Yaskawa INFORM job: A_ROOF_SIDE_0617_2_PAINT_23.JBI

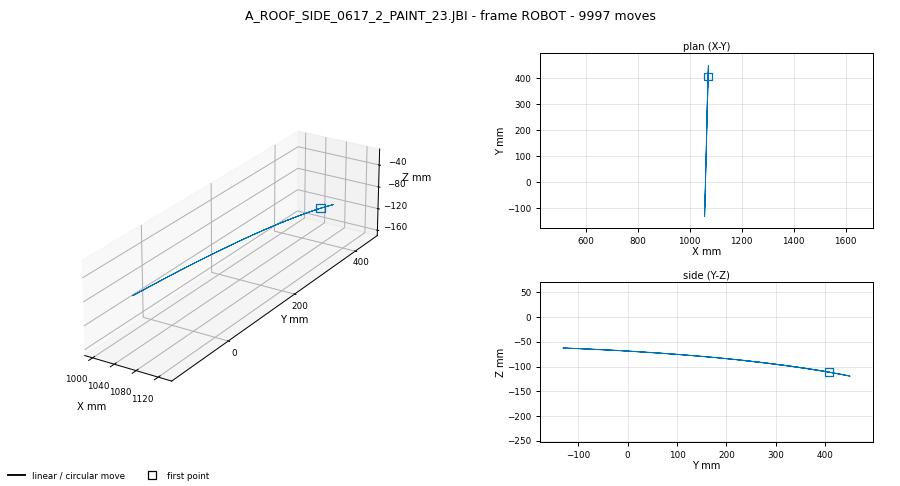
[picture p0: tool path of A_ROOF_SIDE_0617_2_PAINT_23.JBI in frame ROBOT, 9997 of 9997 moves have a stored position in this frame; points joined in program order, loops and branches not executed]
/JOB
//NAME A_ROOF_SIDE_0617_2_PAINT23
//POS
///NPOS 9997,0,0,0,0,0
///TOOL 1
///USER 0
///POSTYPE ROBOT
///RECTAN
///RCONF 1,0,0,0,0,0,0,0,0,0,0,0,0,0,0,0,0,0,0,0,0,0,0,0
C00000=1071.328,407.759,-110.568,175.850,34.121,156.277
C00001=1071.321,407.513,-110.525,175.844,34.112,156.275
C00002=1071.313,407.267,-110.483,175.839,34.102,156.273
C00003=1071.307,407.021,-110.441,175.833,34.094,156.271
C00004=1071.298,406.775,-110.398,175.828,34.084,156.268
C00005=1071.291,406.528,-110.355,175.822,34.075,156.266
C00006=1071.284,406.282,-110.313,175.818,34.066,156.264
C00007=1071.277,406.036,-110.271,175.812,34.057,156.262
C00008=1071.269,405.789,-110.229,175.807,34.048,156.260
C00009=1071.262,405.543,-110.187,175.801,34.039,156.258
C00010=1071.254,405.297,-110.145,175.796,34.030,156.256
C00011=1071.248,405.050,-110.102,175.791,34.021,156.254
C00012=1071.240,404.804,-110.060,175.785,34.012,156.252
C00013=1071.233,404.558,-110.018,175.780,34.003,156.250
C00014=1071.225,404.311,-109.975,175.775,33.995,156.248
C00015=1071.218,404.065,-109.934,175.770,33.986,156.246
C00016=1071.211,403.818,-109.892,175.765,33.977,156.244
C00017=1071.203,403.573,-109.850,175.759,33.968,156.242
C00018=1071.196,403.326,-109.808,175.754,33.959,156.240
C00019=1071.189,403.080,-109.766,175.749,33.951,156.238
C00020=1071.182,402.833,-109.725,175.744,33.942,156.236
C00021=1071.174,402.587,-109.683,175.739,33.933,156.234
C00022=1071.166,402.341,-109.641,175.733,33.925,156.232
C00023=1071.159,402.094,-109.599,175.728,33.916,156.230
C00024=1071.152,401.847,-109.557,175.723,33.907,156.228
C00025=1071.144,401.601,-109.515,175.718,33.899,156.226
C00026=1071.137,401.354,-109.474,175.713,33.890,156.224
C00027=1071.130,401.108,-109.432,175.707,33.882,156.222
C00028=1071.122,400.862,-109.391,175.703,33.873,156.220
C00029=1071.115,400.615,-109.350,175.698,33.865,156.219
C00030=1071.109,400.370,-109.308,175.692,33.856,156.217
C00031=1071.101,400.123,-109.266,175.687,33.848,156.215
C00032=1071.094,399.856,-109.222,175.682,33.838,156.213
C00033=1071.086,399.589,-109.177,175.676,33.829,156.211
C00034=1071.078,399.323,-109.132,175.671,33.820,156.208
C00035=1071.070,399.056,-109.087,175.665,33.811,156.206
C00036=1071.063,398.809,-109.046,175.660,33.803,156.205
C00037=1071.055,398.563,-109.004,175.656,33.794,156.203
C00038=1071.049,398.316,-108.962,175.650,33.786,156.201
C00039=1071.041,398.070,-108.921,175.645,33.778,156.199
C00040=1071.033,397.823,-108.881,175.641,33.770,156.197
C00041=1071.027,397.578,-108.840,175.636,33.761,156.195
C00042=1071.019,397.331,-108.799,175.630,33.753,156.193
C00043=1071.012,397.084,-108.757,175.626,33.745,156.192
C00044=1071.005,396.838,-108.716,175.621,33.737,156.190
C00045=1070.998,396.591,-108.676,175.616,33.729,156.188
C00046=1070.991,396.345,-108.635,175.611,33.720,156.186
C00047=1070.984,396.098,-108.593,175.606,33.712,156.184
C00048=1070.976,395.851,-108.552,175.601,33.704,156.183
C00049=1070.970,395.606,-108.511,175.596,33.696,156.181
C00050=1070.962,395.359,-108.470,175.591,33.688,156.179
C00051=1070.955,395.112,-108.430,175.587,33.680,156.177
C00052=1070.948,394.866,-108.389,175.581,33.672,156.175
C00053=1070.941,394.620,-108.348,175.577,33.664,156.174
C00054=1070.934,394.372,-108.308,175.572,33.656,156.172
C00055=1070.927,394.127,-108.267,175.568,33.648,156.170
C00056=1070.920,393.880,-108.226,175.562,33.640,156.168
C00057=1070.912,393.633,-108.186,175.557,33.632,156.167
C00058=1070.905,393.387,-108.145,175.553,33.624,156.165
C00059=1070.898,393.140,-108.104,175.548,33.617,156.163
C00060=1070.892,392.894,-108.063,175.543,33.608,156.161
C00061=1070.884,392.647,-108.023,175.538,33.600,156.160
C00062=1070.877,392.401,-107.982,175.534,33.593,156.158
C00063=1070.870,392.154,-107.942,175.529,33.585,156.156
C00064=1070.862,391.908,-107.901,175.524,33.578,156.154
C00065=1070.856,391.661,-107.861,175.519,33.570,156.153
C00066=1070.849,391.414,-107.821,175.515,33.562,156.151
C00067=1070.841,391.168,-107.781,175.510,33.554,156.149
C00068=1070.835,390.922,-107.740,175.506,33.546,156.148
C00069=1070.828,390.675,-107.700,175.500,33.539,156.146
C00070=1070.820,390.428,-107.660,175.496,33.531,156.144
C00071=1070.814,390.182,-107.619,175.491,33.523,156.143
C00072=1070.806,389.935,-107.579,175.487,33.516,156.141
C00073=1070.799,389.689,-107.540,175.481,33.508,156.139
C00074=1070.793,389.442,-107.499,175.477,33.501,156.138
C00075=1070.785,389.195,-107.460,175.472,33.493,156.136
C00076=1070.778,388.949,-107.419,175.468,33.486,156.134
C00077=1070.771,388.702,-107.379,175.463,33.478,156.133
C00078=1070.764,388.455,-107.339,175.459,33.471,156.131
C00079=1070.757,388.209,-107.299,175.453,33.463,156.129
C00080=1070.749,387.962,-107.260,175.449,33.456,156.128
C00081=1070.743,387.716,-107.220,175.444,33.448,156.126
C00082=1070.735,387.469,-107.180,175.440,33.441,156.124
C00083=1070.729,387.222,-107.140,175.435,33.433,156.123
C00084=1070.722,386.976,-107.100,175.430,33.426,156.121
C00085=1070.714,386.729,-107.060,175.426,33.419,156.120
C00086=1070.708,386.483,-107.020,175.421,33.411,156.118
C00087=1070.701,386.237,-106.980,175.417,33.404,156.117
C00088=1070.694,385.985,-106.940,175.412,33.396,156.115
C00089=1070.686,385.734,-106.900,175.408,33.389,156.113
C00090=1070.680,385.483,-106.859,175.402,33.382,156.112
C00091=1070.673,385.232,-106.819,175.398,33.374,156.110
C00092=1070.666,384.985,-106.780,175.394,33.367,156.108
C00093=1070.658,384.738,-106.740,175.389,33.360,156.107
C00094=1070.652,384.492,-106.700,175.385,33.352,156.105
C00095=1070.645,384.245,-106.661,175.381,33.345,156.104
C00096=1070.638,383.999,-106.621,175.376,33.338,156.102
C00097=1070.632,383.752,-106.582,175.371,33.331,156.101
C00098=1070.625,383.505,-106.542,175.366,33.323,156.099
C00099=1070.617,383.258,-106.502,175.362,33.316,156.097
C00100=1070.611,383.011,-106.463,175.358,33.309,156.096
C00101=1070.604,382.765,-106.423,175.354,33.302,156.094
C00102=1070.597,382.518,-106.385,175.349,33.295,156.093
C00103=1070.590,382.271,-106.346,175.345,33.288,156.091
C00104=1070.584,382.025,-106.306,175.340,33.281,156.090
C00105=1070.577,381.778,-106.267,175.335,33.274,156.088
C00106=1070.570,381.532,-106.227,175.331,33.266,156.087
C00107=1070.563,381.285,-106.188,175.327,33.260,156.085
C00108=1070.556,381.038,-106.149,175.322,33.252,156.084
C00109=1070.549,380.791,-106.110,175.318,33.245,156.082
C00110=1070.543,380.544,-106.070,175.314,33.239,156.081
C00111=1070.536,380.297,-106.031,175.310,33.232,156.079
C00112=1070.529,380.051,-105.992,175.305,33.225,156.078
C00113=1070.522,379.804,-105.954,175.301,33.217,156.076
C00114=1070.515,379.557,-105.915,175.296,33.211,156.075
C00115=1070.509,379.310,-105.876,175.291,33.204,156.073
C00116=1070.502,379.063,-105.837,175.287,33.197,156.072
C00117=1070.495,378.816,-105.798,175.283,33.190,156.070
C00118=1070.488,378.570,-105.759,175.279,33.183,156.069
C00119=1070.480,378.324,-105.720,175.274,33.176,156.068
C00120=1070.474,378.076,-105.682,175.270,33.170,156.066
C00121=1070.467,377.830,-105.644,175.266,33.163,156.065
C00122=1070.460,377.583,-105.605,175.262,33.156,156.063
C00123=1070.453,377.336,-105.566,175.258,33.149,156.062
C00124=1070.447,377.089,-105.527,175.253,33.143,156.060
C00125=1070.440,376.842,-105.488,175.248,33.136,156.059
C00126=1070.433,376.595,-105.449,175.244,33.129,156.057
C00127=1070.426,376.349,-105.410,175.240,33.122,156.056
C00128=1070.419,376.102,-105.372,175.235,33.115,156.055
C00129=1070.413,375.854,-105.334,175.231,33.109,156.053
C00130=1070.406,375.607,-105.295,175.227,33.102,156.052
C00131=1070.400,375.361,-105.256,175.223,33.096,156.050
C00132=1070.393,375.115,-105.217,175.219,33.089,156.049
C00133=1070.386,374.867,-105.179,175.215,33.082,156.048
C00134=1070.380,374.620,-105.140,175.210,33.075,156.046
C00135=1070.372,374.374,-105.102,175.206,33.069,156.045
C00136=1070.366,374.126,-105.064,175.202,33.062,156.043
C00137=1070.359,373.880,-105.026,175.198,33.055,156.042
C00138=1070.353,373.633,-104.987,175.194,33.049,156.041
C00139=1070.346,373.386,-104.949,175.190,33.042,156.039
C00140=1070.340,373.152,-104.912,175.186,33.037,156.038
C00141=1070.334,372.918,-104.876,175.181,33.030,156.037
C00142=1070.327,372.684,-104.840,175.177,33.024,156.035
C00143=1070.320,372.449,-104.804,175.173,33.018,156.034
C00144=1070.314,372.215,-104.767,175.169,33.012,156.033
C00145=1070.308,371.982,-104.732,175.165,33.006,156.031
C00146=1070.301,371.747,-104.695,175.161,33.000,156.030
C00147=1070.294,371.513,-104.659,175.157,32.993,156.029
C00148=1070.288,371.267,-104.621,175.153,32.987,156.027
C00149=1070.282,371.019,-104.583,175.149,32.981,156.026
C00150=1070.274,370.773,-104.545,175.145,32.974,156.025
C00151=1070.268,370.525,-104.507,175.141,32.968,156.024
C00152=1070.261,370.279,-104.470,175.137,32.962,156.022
C00153=1070.254,370.031,-104.432,175.133,32.955,156.021
C00154=1070.248,369.785,-104.393,175.129,32.949,156.019
C00155=1070.240,369.537,-104.355,175.125,32.942,156.018
C00156=1070.235,369.291,-104.318,175.120,32.936,156.017
C00157=1070.227,369.043,-104.280,175.116,32.930,156.016
C00158=1070.221,368.796,-104.242,175.112,32.924,156.014
C00159=1070.214,368.550,-104.205,175.108,32.917,156.013
C00160=1070.208,368.302,-104.167,175.104,32.911,156.012
C00161=1070.201,368.055,-104.128,175.100,32.905,156.010
C00162=1070.194,367.809,-104.091,175.096,32.898,156.009
C00163=1070.188,367.561,-104.053,175.092,32.892,156.008
C00164=1070.181,367.315,-104.015,175.088,32.886,156.006
C00165=1070.175,367.068,-103.977,175.084,32.880,156.005
C00166=1070.168,366.821,-103.941,175.080,32.874,156.004
C00167=1070.162,366.573,-103.903,175.076,32.867,156.003
C00168=1070.154,366.326,-103.865,175.072,32.861,156.001
C00169=1070.149,366.079,-103.827,175.068,32.855,156.000
C00170=1070.141,365.832,-103.790,175.064,32.849,155.999
C00171=1070.135,365.585,-103.752,175.060,32.842,155.997
C00172=1070.128,365.338,-103.715,175.056,32.837,155.996
C00173=1070.122,365.091,-103.677,175.052,32.830,155.995
C00174=1070.115,364.844,-103.640,175.048,32.824,155.994
C00175=1070.109,364.597,-103.602,175.044,32.818,155.992
C00176=1070.102,364.350,-103.565,175.040,32.812,155.991
C00177=1070.096,364.103,-103.528,175.036,32.806,155.990
C00178=1070.089,363.855,-103.490,175.032,32.800,155.989
C00179=1070.083,363.609,-103.453,175.028,32.794,155.987
C00180=1070.076,363.361,-103.416,175.024,32.788,155.986
C00181=1070.069,363.115,-103.379,175.020,32.782,155.985
C00182=1070.063,362.867,-103.341,175.016,32.776,155.984
C00183=1070.056,362.620,-103.305,175.012,32.770,155.982
C00184=1070.049,362.373,-103.267,175.008,32.764,155.981
C00185=1070.043,362.126,-103.231,175.004,32.758,155.980
C00186=1070.036,361.879,-103.192,175.000,32.752,155.979
C00187=1070.030,361.632,-103.156,174.996,32.746,155.978
C00188=1070.023,361.384,-103.118,174.992,32.740,155.976
C00189=1070.016,361.137,-103.082,174.988,32.734,155.975
C00190=1070.010,360.890,-103.046,174.984,32.728,155.974
C00191=1070.003,360.643,-103.007,174.980,32.722,155.973
C00192=1069.997,360.396,-102.971,174.976,32.716,155.971
C00193=1069.990,360.149,-102.933,174.972,32.710,155.970
C00194=1069.983,359.902,-102.897,174.969,32.705,155.969
C00195=1069.977,359.655,-102.861,174.965,32.699,155.968
C00196=1069.971,359.429,-102.826,174.961,32.694,155.967
C00197=1069.965,359.203,-102.793,174.958,32.688,155.966
C00198=1069.960,358.978,-102.760,174.955,32.683,155.965
C00199=1069.953,358.753,-102.726,174.951,32.677,155.963
C00200=1069.947,358.527,-102.692,174.948,32.672,155.962
C00201=1069.941,358.301,-102.659,174.944,32.667,155.961
C00202=1069.936,358.075,-102.625,174.941,32.661,155.960
C00203=1069.929,357.850,-102.592,174.937,32.656,155.959
C00204=1069.922,357.603,-102.555,174.933,32.651,155.958
C00205=1069.916,357.356,-102.519,174.929,32.645,155.957
C00206=1069.909,357.108,-102.482,174.925,32.639,155.956
C00207=1069.903,356.861,-102.445,174.922,32.633,155.955
C00208=1069.896,356.614,-102.409,174.918,32.628,155.953
C00209=1069.890,356.367,-102.373,174.914,32.622,155.952
C00210=1069.883,356.119,-102.336,174.910,32.616,155.951
C00211=1069.877,355.872,-102.299,174.906,32.610,155.950
C00212=1069.871,355.625,-102.263,174.902,32.605,155.949
C00213=1069.864,355.378,-102.226,174.898,32.599,155.948
C00214=1069.857,355.130,-102.190,174.895,32.594,155.946
C00215=1069.851,354.883,-102.153,174.891,32.588,155.945
C00216=1069.845,354.636,-102.117,174.887,32.582,155.944
C00217=1069.839,354.389,-102.081,174.883,32.576,155.943
C00218=1069.832,354.141,-102.045,174.880,32.571,155.942
C00219=1069.825,353.894,-102.008,174.876,32.565,155.941
C00220=1069.819,353.647,-101.971,174.873,32.560,155.940
C00221=1069.813,353.400,-101.935,174.869,32.554,155.939
C00222=1069.806,353.152,-101.900,174.865,32.548,155.937
C00223=1069.799,352.905,-101.863,174.861,32.543,155.936
C00224=1069.793,352.658,-101.827,174.857,32.537,155.935
C00225=1069.786,352.410,-101.790,174.853,32.532,155.934
C00226=1069.780,352.163,-101.754,174.850,32.526,155.933
C00227=1069.774,351.916,-101.718,174.846,32.521,155.932
C00228=1069.767,351.669,-101.682,174.842,32.515,155.931
C00229=1069.761,351.421,-101.646,174.838,32.509,155.930
C00230=1069.754,351.174,-101.610,174.834,32.504,155.929
C00231=1069.748,350.927,-101.575,174.831,32.499,155.927
C00232=1069.741,350.680,-101.538,174.828,32.493,155.926
C00233=1069.735,350.431,-101.502,174.824,32.488,155.925
C00234=1069.728,350.184,-101.466,174.820,32.482,155.924
C00235=1069.722,349.937,-101.431,174.817,32.477,155.923
C00236=1069.715,349.690,-101.394,174.813,32.471,155.922
C00237=1069.709,349.442,-101.358,174.809,32.466,155.921
C00238=1069.702,349.195,-101.322,174.805,32.460,155.920
C00239=1069.696,348.948,-101.287,174.801,32.455,155.919
C00240=1069.690,348.700,-101.251,174.798,32.450,155.918
C00241=1069.683,348.453,-101.215,174.794,32.444,155.916
C00242=1069.677,348.206,-101.179,174.790,32.439,155.915
C00243=1069.671,347.959,-101.143,174.787,32.433,155.914
C00244=1069.664,347.711,-101.108,174.784,32.428,155.913
C00245=1069.658,347.464,-101.072,174.780,32.423,155.912
C00246=1069.651,347.216,-101.037,174.776,32.417,155.911
C00247=1069.645,346.969,-101.001,174.773,32.412,155.910
C00248=1069.639,346.722,-100.965,174.769,32.407,155.909
C00249=1069.632,346.474,-100.930,174.765,32.401,155.908
C00250=1069.626,346.226,-100.894,174.761,32.396,155.907
C00251=1069.619,345.979,-100.859,174.758,32.391,155.906
C00252=1069.614,345.756,-100.826,174.754,32.386,155.905
C00253=1069.607,345.532,-100.794,174.751,32.381,155.904
C00254=1069.602,345.309,-100.762,174.749,32.376,155.903
C00255=1069.596,345.085,-100.730,174.745,32.371,155.902
C00256=1069.591,344.861,-100.698,174.742,32.366,155.901
C00257=1069.585,344.638,-100.666,174.739,32.362,155.900
C00258=1069.579,344.413,-100.633,174.735,32.357,155.899
C00259=1069.574,344.190,-100.602,174.732,32.352,155.898
C00260=1069.567,343.942,-100.567,174.728,32.347,155.897
C00261=1069.561,343.695,-100.531,174.725,32.341,155.896
C00262=1069.554,343.447,-100.496,174.721,32.337,155.895
C00263=1069.548,343.200,-100.460,174.717,32.331,155.894
C00264=1069.541,342.952,-100.425,174.714,32.326,155.893
C00265=1069.535,342.706,-100.390,174.711,32.320,155.892
C00266=1069.528,342.458,-100.355,174.707,32.316,155.891
C00267=1069.522,342.211,-100.320,174.703,32.310,155.890
C00268=1069.515,341.963,-100.284,174.700,32.305,155.889
C00269=1069.509,341.715,-100.250,174.696,32.300,155.888
C00270=1069.503,341.468,-100.214,174.692,32.295,155.887
C00271=1069.496,341.220,-100.179,174.689,32.289,155.886
C00272=1069.490,340.974,-100.144,174.685,32.285,155.885
C00273=1069.484,340.726,-100.109,174.683,32.279,155.884
C00274=1069.478,340.478,-100.074,174.679,32.274,155.883
C00275=1069.471,340.231,-100.039,174.675,32.269,155.882
C00276=1069.465,339.984,-100.004,174.672,32.264,155.881
C00277=1069.459,339.736,-99.969,174.668,32.259,155.880
C00278=1069.452,339.488,-99.934,174.664,32.254,155.879
C00279=1069.445,339.241,-99.899,174.661,32.248,155.878
C00280=1069.440,338.993,-99.864,174.657,32.243,155.877
C00281=1069.433,338.746,-99.829,174.655,32.238,155.876
C00282=1069.427,338.499,-99.794,174.651,32.233,155.875
C00283=1069.420,338.251,-99.760,174.647,32.228,155.874
C00284=1069.415,338.004,-99.724,174.644,32.223,155.873
C00285=1069.408,337.756,-99.690,174.640,32.218,155.872
C00286=1069.402,337.508,-99.655,174.637,32.213,155.871
C00287=1069.396,337.261,-99.621,174.633,32.208,155.870
C00288=1069.389,337.014,-99.586,174.629,32.203,155.869
C00289=1069.382,336.766,-99.551,174.627,32.198,155.868
C00290=1069.376,336.518,-99.516,174.623,32.193,155.867
C00291=1069.370,336.271,-99.482,174.620,32.188,155.866
C00292=1069.363,336.023,-99.448,174.616,32.183,155.865
C00293=1069.357,335.776,-99.412,174.612,32.178,155.864
C00294=1069.351,335.528,-99.378,174.609,32.173,155.863
C00295=1069.344,335.280,-99.344,174.605,32.168,155.862
C00296=1069.338,335.033,-99.308,174.602,32.163,155.861
C00297=1069.332,334.785,-99.274,174.599,32.158,155.860
C00298=1069.326,334.537,-99.240,174.596,32.153,155.859
C00299=1069.320,334.291,-99.205,174.592,32.148,155.858
C00300=1069.313,334.043,-99.171,174.588,32.143,155.858
C00301=1069.307,333.795,-99.136,174.585,32.138,155.857
C00302=1069.301,333.548,-99.102,174.581,32.133,155.856
C00303=1069.294,333.300,-99.068,174.578,32.128,155.855
C00304=1069.288,333.053,-99.033,174.575,32.123,155.854
C00305=1069.282,332.805,-98.998,174.572,32.118,155.853
C00306=1069.276,332.558,-98.964,174.568,32.113,155.852
C00307=1069.269,332.310,-98.931,174.565,32.109,155.851
C00308=1069.263,332.083,-98.899,174.562,32.104,155.850
C00309=1069.257,331.858,-98.867,174.558,32.099,155.849
C00310=1069.252,331.631,-98.836,174.555,32.095,155.848
C00311=1069.247,331.405,-98.805,174.553,32.091,155.847
C00312=1069.241,331.179,-98.774,174.550,32.086,155.847
C00313=1069.235,330.953,-98.743,174.546,32.082,155.846
C00314=1069.229,330.727,-98.711,174.543,32.077,155.845
C00315=1069.223,330.501,-98.680,174.540,32.073,155.844
C00316=1069.216,330.253,-98.646,174.537,32.068,155.843
C00317=1069.210,330.006,-98.612,174.533,32.063,155.842
C00318=1069.204,329.757,-98.579,174.530,32.058,155.841
C00319=1069.198,329.510,-98.545,174.527,32.054,155.840
C00320=1069.191,329.262,-98.510,174.523,32.049,155.840
C00321=1069.185,329.015,-98.477,174.520,32.045,155.839
C00322=1069.178,328.767,-98.442,174.516,32.040,155.838
C00323=1069.172,328.520,-98.408,174.513,32.035,155.837
C00324=1069.164,328.234,-98.370,174.509,32.029,155.836
C00325=1069.157,327.949,-98.331,174.506,32.024,155.835
C00326=1069.150,327.663,-98.292,174.502,32.019,155.834
C00327=1069.142,327.378,-98.253,174.498,32.013,155.833
C00328=1069.136,327.130,-98.218,174.494,32.008,155.832
C00329=1069.129,326.882,-98.186,174.491,32.003,155.831
C00330=1069.123,326.634,-98.151,174.488,31.999,155.830
C00331=1069.117,326.387,-98.117,174.485,31.994,155.829
C00332=1069.111,326.139,-98.084,174.482,31.989,155.828
C00333=1069.104,325.891,-98.050,174.478,31.985,155.827
C00334=1069.098,325.644,-98.016,174.475,31.980,155.826
C00335=1069.092,325.396,-97.983,174.471,31.975,155.825
C00336=1069.085,325.149,-97.949,174.468,31.971,155.824
C00337=1069.079,324.901,-97.916,174.465,31.966,155.824
C00338=1069.072,324.653,-97.882,174.462,31.961,155.823
C00339=1069.066,324.406,-97.848,174.459,31.957,155.822
C00340=1069.061,324.158,-97.815,174.455,31.952,155.821
C00341=1069.054,323.910,-97.781,174.452,31.947,155.820
C00342=1069.048,323.662,-97.748,174.448,31.943,155.819
C00343=1069.041,323.415,-97.714,174.446,31.938,155.818
C00344=1069.035,323.167,-97.680,174.442,31.933,155.817
C00345=1069.029,322.920,-97.647,174.439,31.929,155.817
C00346=1069.023,322.672,-97.614,174.436,31.924,155.816
C00347=1069.016,322.424,-97.580,174.432,31.919,155.815
C00348=1069.010,322.176,-97.546,174.429,31.915,155.814
C00349=1069.004,321.929,-97.514,174.426,31.910,155.813
C00350=1068.998,321.681,-97.480,174.423,31.905,155.812
C00351=1068.991,321.433,-97.447,174.420,31.901,155.811
C00352=1068.986,321.185,-97.413,174.416,31.896,155.810
C00353=1068.979,320.938,-97.380,174.413,31.891,155.809
C00354=1068.974,320.690,-97.346,174.410,31.887,155.809
C00355=1068.967,320.443,-97.314,174.407,31.882,155.808
C00356=1068.961,320.194,-97.280,174.404,31.878,155.807
C00357=1068.955,319.947,-97.246,174.400,31.873,155.806
C00358=1068.948,319.700,-97.214,174.397,31.868,155.805
C00359=1068.943,319.452,-97.180,174.394,31.864,155.804
C00360=1068.936,319.204,-97.148,174.391,31.859,155.803
C00361=1068.931,318.957,-97.114,174.388,31.855,155.803
C00362=1068.924,318.708,-97.080,174.385,31.850,155.802
C00363=1068.918,318.461,-97.047,174.381,31.845,155.801
C00364=1068.913,318.251,-97.019,174.378,31.841,155.800
C00365=1068.907,318.041,-96.991,174.376,31.838,155.799
C00366=1068.903,317.830,-96.963,174.374,31.833,155.799
C00367=1068.898,317.620,-96.935,174.371,31.830,155.798
C00368=1068.892,317.410,-96.907,174.368,31.825,155.797
C00369=1068.888,317.199,-96.879,174.365,31.822,155.796
C00370=1068.882,316.989,-96.851,174.362,31.817,155.796
C00371=1068.877,316.779,-96.823,174.360,31.814,155.795
C00372=1068.871,316.531,-96.790,174.357,31.809,155.794
C00373=1068.865,316.283,-96.757,174.354,31.805,155.793
C00374=1068.859,316.036,-96.724,174.351,31.800,155.792
C00375=1068.853,315.788,-96.691,174.347,31.795,155.791
C00376=1068.847,315.540,-96.658,174.344,31.791,155.791
C00377=1068.841,315.293,-96.625,174.341,31.786,155.790
C00378=1068.835,315.045,-96.592,174.338,31.781,155.789
C00379=1068.829,314.797,-96.559,174.335,31.777,155.788
C00380=1068.823,314.549,-96.526,174.332,31.772,155.787
C00381=1068.817,314.302,-96.493,174.329,31.768,155.786
C00382=1068.811,314.053,-96.461,174.325,31.764,155.785
C00383=1068.804,313.805,-96.428,174.323,31.759,155.785
C00384=1068.798,313.558,-96.395,174.320,31.755,155.784
C00385=1068.791,313.310,-96.362,174.316,31.750,155.783
C00386=1068.785,313.062,-96.330,174.313,31.746,155.782
C00387=1068.779,312.814,-96.298,174.310,31.742,155.781
C00388=1068.773,312.567,-96.265,174.307,31.737,155.781
C00389=1068.766,312.319,-96.233,174.304,31.733,155.780
C00390=1068.760,312.071,-96.201,174.301,31.728,155.779
C00391=1068.754,311.823,-96.168,174.297,31.724,155.778
C00392=1068.747,311.576,-96.135,174.294,31.719,155.777
C00393=1068.741,311.328,-96.103,174.291,31.715,155.776
C00394=1068.735,311.080,-96.070,174.289,31.711,155.776
C00395=1068.729,310.833,-96.038,174.285,31.706,155.775
C00396=1068.723,310.584,-96.006,174.282,31.702,155.774
C00397=1068.716,310.337,-95.973,174.279,31.697,155.773
C00398=1068.709,310.089,-95.941,174.275,31.693,155.772
C00399=1068.703,309.841,-95.909,174.273,31.689,155.772
C00400=1068.697,309.594,-95.876,174.270,31.684,155.771
C00401=1068.691,309.345,-95.844,174.267,31.680,155.770
C00402=1068.685,309.098,-95.811,174.263,31.676,155.769
C00403=1068.679,308.850,-95.779,174.260,31.671,155.768
C00404=1068.672,308.602,-95.747,174.258,31.667,155.768
C00405=1068.666,308.354,-95.715,174.255,31.663,155.767
C00406=1068.660,308.107,-95.682,174.251,31.658,155.766
C00407=1068.654,307.859,-95.651,174.248,31.654,155.765
C00408=1068.648,307.611,-95.618,174.245,31.649,155.764
C00409=1068.642,307.363,-95.586,174.243,31.645,155.764
C00410=1068.635,307.115,-95.554,174.239,31.641,155.763
C00411=1068.629,306.868,-95.522,174.236,31.636,155.762
C00412=1068.623,306.619,-95.490,174.233,31.632,155.761
C00413=1068.617,306.372,-95.457,174.230,31.628,155.760
C00414=1068.611,306.124,-95.425,174.227,31.623,155.760
C00415=1068.604,305.876,-95.394,174.224,31.619,155.759
C00416=1068.598,305.629,-95.361,174.221,31.615,155.758
C00417=1068.592,305.381,-95.329,174.218,31.610,155.757
C00418=1068.586,305.132,-95.297,174.215,31.606,155.756
C00419=1068.580,304.885,-95.266,174.212,31.602,155.756
C00420=1068.575,304.658,-95.236,174.209,31.597,155.755
C00421=1068.569,304.430,-95.207,174.206,31.594,155.754
C00422=1068.564,304.203,-95.177,174.203,31.589,155.753
C00423=1068.558,303.975,-95.148,174.201,31.586,155.753
C00424=1068.552,303.748,-95.119,174.199,31.581,155.752
C00425=1068.547,303.521,-95.090,174.196,31.578,155.751
C00426=1068.541,303.293,-95.060,174.193,31.573,155.750
C00427=1068.535,303.066,-95.031,174.190,31.570,155.750
C00428=1068.529,302.817,-94.999,174.187,31.565,155.749
C00429=1068.523,302.569,-94.967,174.184,31.561,155.748
C00430=1068.518,302.322,-94.935,174.181,31.557,155.747
C00431=1068.511,302.074,-94.904,174.178,31.552,155.747
C00432=1068.505,301.826,-94.871,174.175,31.548,155.746
C00433=1068.499,301.579,-94.840,174.173,31.544,155.745
C00434=1068.493,301.331,-94.808,174.169,31.539,155.744
C00435=1068.487,301.083,-94.776,174.166,31.535,155.743
C00436=1068.481,300.835,-94.744,174.163,31.531,155.743
C00437=1068.475,300.587,-94.712,174.160,31.526,155.742
C00438=1068.469,300.339,-94.681,174.158,31.522,155.741
C00439=1068.463,300.092,-94.649,174.155,31.518,155.740
C00440=1068.457,299.843,-94.617,174.152,31.514,155.739
C00441=1068.451,299.596,-94.586,174.148,31.509,155.739
C00442=1068.445,299.348,-94.554,174.146,31.505,155.738
C00443=1068.440,299.099,-94.523,174.143,31.500,155.737
C00444=1068.433,298.852,-94.492,174.140,31.496,155.736
C00445=1068.427,298.604,-94.460,174.137,31.492,155.735
C00446=1068.422,298.356,-94.428,174.134,31.488,155.735
C00447=1068.415,298.108,-94.397,174.132,31.483,155.734
C00448=1068.410,297.861,-94.365,174.128,31.479,155.733
C00449=1068.404,297.612,-94.333,174.125,31.474,155.732
C00450=1068.397,297.364,-94.302,174.122,31.470,155.731
C00451=1068.392,297.116,-94.271,174.120,31.466,155.731
C00452=1068.385,296.869,-94.239,174.117,31.462,155.730
C00453=1068.380,296.621,-94.208,174.114,31.457,155.729
C00454=1068.374,296.373,-94.177,174.111,31.453,155.728
C00455=1068.368,296.124,-94.145,174.108,31.449,155.728
C00456=1068.361,295.877,-94.114,174.105,31.445,155.727
C00457=1068.355,295.629,-94.083,174.102,31.440,155.726
C00458=1068.350,295.381,-94.051,174.099,31.436,155.725
C00459=1068.343,295.133,-94.020,174.096,31.432,155.725
C00460=1068.337,294.885,-93.990,174.094,31.428,155.724
C00461=1068.331,294.637,-93.958,174.091,31.424,155.723
C00462=1068.325,294.389,-93.927,174.088,31.419,155.722
C00463=1068.319,294.141,-93.896,174.085,31.416,155.722
C00464=1068.313,293.893,-93.864,174.082,31.411,155.721
C00465=1068.307,293.645,-93.833,174.079,31.407,155.720
C00466=1068.300,293.397,-93.802,174.076,31.402,155.719
C00467=1068.294,293.150,-93.772,174.073,31.399,155.719
C00468=1068.288,292.901,-93.740,174.070,31.394,155.718
C00469=1068.282,292.654,-93.709,174.068,31.390,155.717
C00470=1068.276,292.406,-93.678,174.065,31.386,155.716
C00471=1068.270,292.158,-93.647,174.062,31.382,155.716
C00472=1068.264,291.910,-93.615,174.059,31.378,155.715
C00473=1068.258,291.662,-93.585,174.057,31.373,155.714
C00474=1068.252,291.413,-93.554,174.054,31.370,155.713
C00475=1068.246,291.166,-93.523,174.051,31.365,155.712
C00476=1068.240,290.946,-93.496,174.048,31.361,155.712
C00477=1068.235,290.726,-93.468,174.045,31.358,155.711
C00478=1068.230,290.505,-93.441,174.044,31.354,155.710
C00479=1068.225,290.285,-93.414,174.041,31.350,155.710
C00480=1068.219,290.066,-93.386,174.038,31.346,155.709
C00481=1068.214,289.846,-93.359,174.035,31.343,155.708
C00482=1068.208,289.626,-93.332,174.034,31.339,155.708
C00483=1068.203,289.405,-93.304,174.031,31.336,155.707
C00484=1068.197,289.158,-93.274,174.028,31.332,155.706
C00485=1068.191,288.910,-93.242,174.025,31.327,155.706
C00486=1068.185,288.662,-93.212,174.022,31.323,155.705
C00487=1068.178,288.413,-93.181,174.020,31.319,155.704
C00488=1068.173,288.165,-93.151,174.017,31.315,155.703
C00489=1068.166,287.917,-93.120,174.014,31.311,155.703
C00490=1068.160,287.670,-93.089,174.011,31.307,155.702
C00491=1068.154,287.422,-93.059,174.009,31.303,155.701
C00492=1068.148,287.173,-93.028,174.006,31.299,155.700
C00493=1068.142,286.926,-92.998,174.003,31.294,155.700
C00494=1068.136,286.677,-92.967,174.000,31.290,155.699
C00495=1068.130,286.429,-92.937,173.997,31.286,155.698
C00496=1068.124,286.181,-92.906,173.994,31.282,155.698
C00497=1068.117,285.933,-92.876,173.991,31.278,155.697
C00498=1068.112,285.685,-92.845,173.988,31.274,155.696
C00499=1068.106,285.437,-92.815,173.986,31.270,155.695
C00500=1068.099,285.189,-92.784,173.983,31.265,155.695
C00501=1068.094,284.941,-92.754,173.980,31.262,155.694
C00502=1068.088,284.693,-92.723,173.977,31.257,155.693
C00503=1068.081,284.445,-92.693,173.975,31.253,155.692
C00504=1068.076,284.197,-92.662,173.972,31.249,155.692
C00505=1068.069,283.949,-92.633,173.969,31.245,155.691
C00506=1068.063,283.701,-92.602,173.966,31.241,155.690
C00507=1068.057,283.453,-92.572,173.964,31.237,155.689
C00508=1068.051,283.205,-92.541,173.961,31.233,155.689
C00509=1068.045,282.957,-92.510,173.958,31.228,155.688
C00510=1068.039,282.709,-92.480,173.955,31.225,155.687
C00511=1068.033,282.461,-92.450,173.953,31.220,155.686
C00512=1068.027,282.212,-92.420,173.950,31.216,155.686
C00513=1068.021,281.964,-92.389,173.948,31.212,155.685
C00514=1068.015,281.716,-92.359,173.945,31.208,155.684
C00515=1068.009,281.468,-92.329,173.943,31.204,155.684
C00516=1068.003,281.221,-92.299,173.940,31.200,155.683
C00517=1067.997,280.972,-92.269,173.937,31.196,155.682
C00518=1067.991,280.724,-92.239,173.934,31.192,155.681
C00519=1067.985,280.476,-92.208,173.932,31.187,155.681
C00520=1067.979,280.228,-92.178,173.929,31.184,155.680
C00521=1067.974,279.980,-92.148,173.926,31.180,155.679
C00522=1067.967,279.732,-92.118,173.923,31.175,155.678
C00523=1067.961,279.484,-92.088,173.921,31.172,155.678
C00524=1067.955,279.235,-92.058,173.918,31.167,155.677
C00525=1067.949,278.988,-92.028,173.915,31.163,155.676
C00526=1067.942,278.739,-91.998,173.912,31.159,155.676
C00527=1067.937,278.491,-91.968,173.910,31.155,155.675
C00528=1067.930,278.243,-91.938,173.907,31.151,155.674
C00529=1067.925,277.995,-91.909,173.904,31.147,155.673
C00530=1067.919,277.747,-91.878,173.901,31.143,155.673
C00531=1067.913,277.499,-91.848,173.899,31.139,155.672
C00532=1067.907,277.284,-91.822,173.897,31.135,155.671
C00533=1067.902,277.069,-91.797,173.894,31.132,155.671
C00534=1067.897,276.854,-91.771,173.892,31.128,155.670
C00535=1067.891,276.639,-91.745,173.890,31.125,155.669
C00536=1067.886,276.425,-91.719,173.888,31.121,155.669
C00537=1067.881,276.209,-91.693,173.885,31.118,155.668
C00538=1067.876,275.995,-91.668,173.883,31.115,155.668
C00539=1067.870,275.780,-91.642,173.880,31.111,155.667
C00540=1067.865,275.531,-91.612,173.878,31.107,155.666
C00541=1067.859,275.284,-91.582,173.875,31.103,155.666
C00542=1067.853,275.036,-91.553,173.872,31.099,155.665
C00543=1067.847,274.787,-91.523,173.870,31.094,155.664
C00544=1067.841,274.540,-91.493,173.867,31.091,155.663
C00545=1067.835,274.291,-91.463,173.865,31.086,155.663
C00546=1067.829,274.043,-91.434,173.862,31.083,155.662
C00547=1067.822,273.794,-91.404,173.860,31.078,155.661
C00548=1067.817,273.546,-91.374,173.857,31.074,155.660
C00549=1067.811,273.298,-91.345,173.854,31.071,155.660
C00550=1067.805,273.050,-91.315,173.851,31.066,155.659
C00551=1067.799,272.802,-91.286,173.849,31.062,155.658
C00552=1067.793,272.554,-91.256,173.846,31.058,155.658
C00553=1067.787,272.305,-91.227,173.843,31.054,155.657
C00554=1067.780,272.058,-91.197,173.840,31.050,155.656
C00555=1067.775,271.809,-91.168,173.839,31.046,155.655
C00556=1067.769,271.561,-91.139,173.836,31.042,155.655
C00557=1067.763,271.313,-91.109,173.833,31.038,155.654
C00558=1067.756,271.065,-91.079,173.831,31.034,155.653
C00559=1067.751,270.817,-91.050,173.828,31.030,155.653
C00560=1067.745,270.569,-91.021,173.825,31.026,155.652
C00561=1067.738,270.321,-90.991,173.822,31.022,155.651
C00562=1067.733,270.072,-90.962,173.820,31.018,155.650
C00563=1067.727,269.824,-90.933,173.818,31.014,155.650
C00564=1067.721,269.576,-90.903,173.815,31.010,155.649
C00565=1067.715,269.327,-90.874,173.812,31.006,155.648
C00566=1067.709,269.079,-90.845,173.810,31.002,155.648
C00567=1067.703,268.831,-90.815,173.807,30.998,155.647
C00568=1067.697,268.583,-90.786,173.804,30.994,155.646
C00569=1067.691,268.335,-90.757,173.802,30.990,155.646
C00570=1067.684,268.087,-90.728,173.800,30.986,155.645
C00571=1067.679,267.838,-90.699,173.797,30.982,155.644
C00572=1067.673,267.590,-90.670,173.794,30.978,155.644
C00573=1067.666,267.342,-90.641,173.792,30.974,155.643
C00574=1067.660,267.094,-90.612,173.789,30.970,155.642
C00575=1067.655,266.845,-90.582,173.786,30.966,155.641
C00576=1067.648,266.597,-90.553,173.783,30.962,155.641
C00577=1067.642,266.349,-90.524,173.782,30.958,155.640
C00578=1067.636,266.101,-90.495,173.779,30.954,155.639
C00579=1067.630,265.852,-90.465,173.776,30.950,155.639
C00580=1067.624,265.604,-90.436,173.774,30.946,155.638
C00581=1067.618,265.356,-90.407,173.771,30.942,155.637
C00582=1067.612,265.107,-90.379,173.769,30.938,155.636
C00583=1067.606,264.859,-90.349,173.766,30.934,155.636
C00584=1067.600,264.611,-90.320,173.764,30.930,155.635
C00585=1067.594,264.363,-90.291,173.761,30.926,155.634
C00586=1067.588,264.115,-90.262,173.758,30.922,155.634
C00587=1067.582,263.867,-90.234,173.756,30.918,155.633
C00588=1067.578,263.653,-90.208,173.754,30.915,155.632
C00589=1067.572,263.440,-90.183,173.752,30.911,155.632
C00590=1067.567,263.227,-90.159,173.749,30.908,155.631
C00591=1067.561,263.014,-90.134,173.748,30.904,155.631
C00592=1067.556,262.801,-90.110,173.745,30.901,155.630
C00593=1067.551,262.588,-90.085,173.743,30.898,155.629
C00594=1067.545,262.374,-90.061,173.741,30.894,155.629
C00595=1067.540,262.162,-90.036,173.739,30.891,155.628
C00596=1067.534,261.914,-90.007,173.736,30.887,155.627
C00597=1067.528,261.665,-89.979,173.733,30.883,155.627
C00598=1067.522,261.417,-89.950,173.731,30.879,155.626
C00599=1067.516,261.168,-89.921,173.729,30.875,155.625
C00600=1067.510,260.920,-89.892,173.726,30.871,155.625
C00601=1067.504,260.671,-89.864,173.723,30.867,155.624
C00602=1067.497,260.423,-89.835,173.721,30.863,155.623
C00603=1067.491,260.175,-89.806,173.719,30.860,155.623
C00604=1067.485,259.927,-89.778,173.716,30.855,155.622
C00605=1067.479,259.679,-89.749,173.713,30.851,155.621
C00606=1067.473,259.430,-89.721,173.711,30.848,155.621
C00607=1067.467,259.182,-89.692,173.709,30.844,155.620
C00608=1067.461,258.933,-89.664,173.706,30.839,155.619
C00609=1067.455,258.685,-89.635,173.704,30.836,155.618
C00610=1067.449,258.438,-89.607,173.701,30.832,155.618
C00611=1067.443,258.189,-89.579,173.698,30.828,155.617
C00612=1067.436,257.941,-89.550,173.696,30.824,155.616
C00613=1067.430,257.692,-89.522,173.694,30.820,155.616
C00614=1067.424,257.444,-89.493,173.691,30.816,155.615
C00615=1067.419,257.196,-89.465,173.688,30.812,155.614
C00616=1067.413,256.947,-89.436,173.687,30.808,155.614
C00617=1067.406,256.699,-89.408,173.684,30.804,155.613
C00618=1067.400,256.450,-89.380,173.681,30.800,155.612
C00619=1067.394,256.202,-89.351,173.678,30.796,155.612
C00620=1067.388,255.954,-89.323,173.677,30.792,155.611
C00621=1067.382,255.706,-89.294,173.674,30.788,155.610
C00622=1067.376,255.457,-89.266,173.671,30.784,155.610
C00623=1067.370,255.210,-89.238,173.669,30.780,155.609
C00624=1067.364,254.961,-89.209,173.667,30.776,155.608
C00625=1067.358,254.712,-89.181,173.664,30.772,155.607
C00626=1067.352,254.463,-89.153,173.662,30.769,155.607
C00627=1067.347,254.216,-89.124,173.659,30.764,155.606
C00628=1067.340,253.968,-89.096,173.657,30.760,155.605
C00629=1067.334,253.719,-89.068,173.654,30.757,155.605
C00630=1067.329,253.471,-89.040,173.652,30.752,155.604
C00631=1067.323,253.222,-89.012,173.650,30.749,155.603
C00632=1067.316,252.974,-88.983,173.647,30.745,155.603
C00633=1067.310,252.726,-88.955,173.645,30.740,155.602
C00634=1067.304,252.477,-88.927,173.642,30.736,155.601
C00635=1067.298,252.229,-88.899,173.640,30.733,155.600
C00636=1067.293,251.981,-88.871,173.638,30.728,155.600
C00637=1067.286,251.732,-88.843,173.635,30.724,155.599
C00638=1067.281,251.484,-88.815,173.633,30.721,155.598
C00639=1067.275,251.235,-88.787,173.631,30.716,155.598
C00640=1067.269,250.987,-88.758,173.628,30.712,155.597
C00641=1067.263,250.739,-88.731,173.625,30.709,155.596
C00642=1067.257,250.490,-88.703,173.624,30.704,155.596
C00643=1067.252,250.242,-88.675,173.621,30.700,155.595
C00644=1067.246,250.028,-88.650,173.619,30.697,155.594
C00645=1067.241,249.814,-88.627,173.616,30.693,155.594
C00646=1067.236,249.599,-88.601,173.615,30.690,155.593
C00647=1067.231,249.385,-88.578,173.613,30.687,155.592
C00648=1067.226,249.171,-88.554,173.611,30.683,155.592
C00649=1067.221,248.956,-88.529,173.608,30.680,155.591
C00650=1067.216,248.742,-88.505,173.607,30.676,155.591
C00651=1067.211,248.527,-88.481,173.605,30.673,155.590
C00652=1067.205,248.279,-88.454,173.602,30.669,155.589
C00653=1067.199,248.031,-88.426,173.600,30.665,155.589
C00654=1067.193,247.783,-88.398,173.598,30.661,155.588
C00655=1067.187,247.534,-88.370,173.595,30.656,155.587
C00656=1067.182,247.286,-88.342,173.593,30.653,155.586
C00657=1067.175,247.038,-88.314,173.591,30.649,155.586
C00658=1067.170,246.789,-88.286,173.588,30.644,155.585
C00659=1067.164,246.540,-88.258,173.586,30.641,155.584
C00660=1067.158,246.292,-88.231,173.584,30.636,155.584
C00661=1067.152,246.044,-88.203,173.581,30.632,155.583
C00662=1067.146,245.796,-88.175,173.578,30.629,155.582
C00663=1067.140,245.547,-88.147,173.577,30.625,155.582
C00664=1067.135,245.299,-88.120,173.574,30.620,155.581
C00665=1067.129,245.050,-88.092,173.571,30.616,155.580
C00666=1067.123,244.802,-88.065,173.570,30.613,155.580
C00667=1067.117,244.553,-88.037,173.567,30.608,155.579
C00668=1067.111,244.305,-88.010,173.564,30.604,155.578
C00669=1067.104,244.057,-87.982,173.563,30.601,155.577
C00670=1067.099,243.809,-87.954,173.560,30.596,155.577
C00671=1067.092,243.560,-87.927,173.557,30.592,155.576
C00672=1067.087,243.312,-87.899,173.556,30.589,155.575
C00673=1067.081,243.062,-87.872,173.553,30.584,155.575
C00674=1067.075,242.814,-87.844,173.551,30.581,155.574
C00675=1067.069,242.567,-87.817,173.549,30.577,155.573
C00676=1067.064,242.317,-87.789,173.546,30.572,155.572
C00677=1067.058,242.070,-87.762,173.544,30.569,155.572
C00678=1067.051,241.821,-87.735,173.542,30.565,155.571
C00679=1067.045,241.573,-87.707,173.539,30.561,155.571
C00680=1067.039,241.323,-87.680,173.537,30.557,155.570
C00681=1067.033,241.076,-87.652,173.535,30.553,155.569
C00682=1067.027,240.827,-87.625,173.533,30.549,155.568
C00683=1067.021,240.579,-87.598,173.530,30.545,155.568
C00684=1067.015,240.330,-87.570,173.528,30.541,155.567
C00685=1067.009,240.082,-87.543,173.526,30.537,155.566
C00686=1067.003,239.833,-87.516,173.523,30.533,155.566
C00687=1066.997,239.585,-87.489,173.521,30.529,155.565
C00688=1066.992,239.336,-87.461,173.519,30.525,155.564
C00689=1066.985,239.088,-87.434,173.516,30.521,155.564
C00690=1066.979,238.839,-87.407,173.515,30.517,155.563
C00691=1066.973,238.590,-87.380,173.512,30.513,155.562
C00692=1066.967,238.343,-87.353,173.509,30.509,155.561
C00693=1066.962,238.094,-87.325,173.508,30.505,155.561
C00694=1066.955,237.845,-87.298,173.505,30.501,155.560
C00695=1066.949,237.597,-87.271,173.503,30.497,155.559
C00696=1066.943,237.348,-87.244,173.501,30.493,155.559
C00697=1066.937,237.100,-87.217,173.498,30.489,155.558
C00698=1066.931,236.852,-87.190,173.496,30.485,155.557
C00699=1066.925,236.603,-87.162,173.494,30.481,155.557
C00700=1066.921,236.386,-87.139,173.492,30.478,155.556
C00701=1066.915,236.168,-87.116,173.490,30.474,155.555
C00702=1066.910,235.951,-87.092,173.489,30.471,155.555
C00703=1066.905,235.733,-87.068,173.486,30.467,155.554
C00704=1066.900,235.516,-87.045,173.484,30.463,155.554
C00705=1066.894,235.298,-87.021,173.482,30.460,155.553
C00706=1066.889,235.080,-86.997,173.481,30.457,155.552
C00707=1066.884,234.863,-86.974,173.478,30.453,155.552
C00708=1066.878,234.615,-86.946,173.476,30.449,155.551
C00709=1066.872,234.366,-86.919,173.474,30.445,155.550
C00710=1066.866,234.118,-86.893,173.472,30.441,155.550
C00711=1066.860,233.870,-86.866,173.469,30.437,155.549
C00712=1066.855,233.621,-86.839,173.467,30.433,155.548
C00713=1066.848,233.372,-86.812,173.465,30.429,155.548
C00714=1066.842,233.124,-86.785,173.462,30.425,155.547
C00715=1066.836,232.876,-86.758,173.461,30.421,155.546
C00716=1066.830,232.627,-86.731,173.458,30.417,155.546
C00717=1066.824,232.379,-86.705,173.456,30.413,155.545
C00718=1066.818,232.130,-86.678,173.454,30.409,155.544
C00719=1066.813,231.882,-86.651,173.452,30.405,155.543
C00720=1066.806,231.633,-86.624,173.450,30.401,155.543
C00721=1066.800,231.384,-86.598,173.448,30.397,155.542
C00722=1066.795,231.136,-86.571,173.445,30.393,155.541
C00723=1066.789,230.888,-86.544,173.443,30.389,155.541
C00724=1066.783,230.639,-86.517,173.441,30.385,155.540
C00725=1066.777,230.390,-86.491,173.438,30.381,155.539
C00726=1066.771,230.142,-86.464,173.437,30.377,155.538
C00727=1066.765,229.894,-86.437,173.434,30.373,155.538
C00728=1066.759,229.645,-86.411,173.432,30.369,155.537
C00729=1066.753,229.396,-86.384,173.430,30.365,155.536
C00730=1066.748,229.147,-86.358,173.428,30.361,155.536
C00731=1066.742,228.899,-86.331,173.425,30.357,155.535
C00732=1066.735,228.650,-86.305,173.424,30.353,155.534
C00733=1066.729,228.402,-86.278,173.421,30.349,155.534
C00734=1066.723,228.153,-86.251,173.419,30.345,155.533
C00735=1066.717,227.905,-86.225,173.417,30.341,155.532
C00736=1066.711,227.657,-86.199,173.415,30.337,155.532
C00737=1066.705,227.407,-86.172,173.413,30.333,155.531
C00738=1066.699,227.159,-86.146,173.411,30.329,155.530
C00739=1066.693,226.911,-86.119,173.408,30.325,155.530
C00740=1066.687,226.662,-86.093,173.407,30.321,155.529
C00741=1066.681,226.414,-86.066,173.404,30.317,155.528
C00742=1066.675,226.165,-86.041,173.402,30.314,155.528
C00743=1066.669,225.916,-86.014,173.400,30.309,155.527
C00744=1066.663,225.668,-85.987,173.398,30.305,155.526
C00745=1066.657,225.419,-85.962,173.395,30.301,155.525
C00746=1066.651,225.171,-85.935,173.394,30.297,155.525
C00747=1066.646,224.922,-85.908,173.391,30.293,155.524
C00748=1066.639,224.674,-85.882,173.389,30.289,155.523
C00749=1066.634,224.425,-85.856,173.387,30.285,155.523
C00750=1066.628,224.177,-85.830,173.385,30.281,155.522
C00751=1066.621,223.928,-85.803,173.383,30.277,155.521
C00752=1066.615,223.679,-85.777,173.381,30.273,155.520
C00753=1066.609,223.431,-85.751,173.378,30.269,155.520
C00754=1066.604,223.182,-85.725,173.377,30.265,155.519
C00755=1066.598,222.934,-85.698,173.374,30.261,155.518
C00756=1066.593,222.712,-85.676,173.372,30.257,155.518
C00757=1066.587,222.491,-85.652,173.371,30.253,155.517
C00758=1066.582,222.269,-85.629,173.369,30.250,155.517
C00759=1066.577,222.048,-85.606,173.366,30.246,155.516
C00760=1066.571,221.826,-85.581,173.365,30.243,155.515
C00761=1066.566,221.605,-85.558,173.363,30.239,155.515
C00762=1066.561,221.383,-85.535,173.361,30.236,155.514
C00763=1066.556,221.161,-85.512,173.360,30.232,155.513
C00764=1066.549,220.913,-85.486,173.357,30.228,155.513
C00765=1066.544,220.664,-85.460,173.355,30.224,155.512
C00766=1066.537,220.416,-85.434,173.353,30.220,155.511
C00767=1066.532,220.167,-85.408,173.351,30.216,155.511
C00768=1066.525,219.919,-85.382,173.349,30.212,155.510
C00769=1066.520,219.670,-85.356,173.347,30.208,155.509
C00770=1066.513,219.422,-85.330,173.344,30.204,155.509
C00771=1066.508,219.173,-85.304,173.343,30.200,155.508
C00772=1066.502,218.924,-85.279,173.341,30.196,155.507
C00773=1066.496,218.676,-85.252,173.338,30.192,155.506
C00774=1066.490,218.427,-85.227,173.337,30.188,155.506
C00775=1066.483,218.179,-85.201,173.334,30.184,155.505
C00776=1066.478,217.930,-85.175,173.333,30.180,155.504
C00777=1066.472,217.682,-85.149,173.330,30.175,155.504
C00778=1066.466,217.433,-85.123,173.328,30.172,155.503
C00779=1066.460,217.185,-85.097,173.327,30.167,155.502
C00780=1066.454,216.936,-85.072,173.324,30.163,155.502
C00781=1066.448,216.687,-85.046,173.322,30.160,155.501
C00782=1066.442,216.439,-85.020,173.320,30.155,155.500
C00783=1066.436,216.190,-84.994,173.318,30.151,155.499
C00784=1066.430,215.941,-84.969,173.316,30.147,155.499
C00785=1066.424,215.692,-84.943,173.314,30.143,155.498
C00786=1066.418,215.444,-84.917,173.312,30.139,155.497
C00787=1066.412,215.195,-84.891,173.310,30.135,155.497
C00788=1066.406,214.947,-84.866,173.308,30.131,155.496
C00789=1066.401,214.698,-84.840,173.306,30.127,155.495
C00790=1066.394,214.450,-84.814,173.304,30.123,155.495
C00791=1066.388,214.201,-84.788,173.301,30.118,155.494
C00792=1066.383,213.953,-84.763,173.300,30.115,155.493
C00793=1066.377,213.704,-84.737,173.298,30.110,155.492
C00794=1066.371,213.455,-84.711,173.296,30.106,155.492
C00795=1066.365,213.206,-84.686,173.294,30.102,155.491
C00796=1066.359,212.958,-84.661,173.291,30.098,155.490
C00797=1066.354,212.709,-84.635,173.290,30.094,155.489
C00798=1066.347,212.461,-84.609,173.288,30.090,155.489
C00799=1066.341,212.212,-84.583,173.285,30.086,155.488
C00800=1066.335,211.963,-84.558,173.284,30.082,155.487
C00801=1066.330,211.715,-84.533,173.282,30.078,155.487
C00802=1066.324,211.466,-84.507,173.280,30.074,155.486
C00803=1066.317,211.218,-84.482,173.278,30.070,155.485
C00804=1066.311,210.969,-84.457,173.275,30.065,155.485
C00805=1066.306,210.720,-84.431,173.274,30.062,155.484
C00806=1066.299,210.471,-84.405,173.272,30.057,155.483
C00807=1066.293,210.223,-84.380,173.270,30.053,155.482
C00808=1066.287,209.974,-84.355,173.268,30.050,155.482
C00809=1066.281,209.726,-84.330,173.265,30.045,155.481
C00810=1066.276,209.477,-84.304,173.264,30.041,155.480
C00811=1066.270,209.228,-84.278,173.262,30.037,155.480
C00812=1066.264,209.010,-84.257,173.261,30.034,155.479
C00813=1066.259,208.790,-84.234,173.258,30.030,155.478
C00814=1066.253,208.571,-84.212,173.256,30.026,155.478
C00815=1066.249,208.352,-84.190,173.255,30.022,155.477
C00816=1066.244,208.133,-84.167,173.253,30.019,155.477
C00817=1066.238,207.913,-84.145,173.251,30.015,155.476
C00818=1066.233,207.694,-84.123,173.250,30.012,155.475
C00819=1066.228,207.475,-84.101,173.248,30.008,155.475
C00820=1066.203,206.430,-83.998,173.094,29.931,155.470
C00821=1066.197,206.180,-83.973,173.091,29.928,155.469
C00822=1066.192,205.932,-83.949,173.089,29.925,155.469
C00823=1066.186,205.683,-83.925,173.087,29.922,155.468
C00824=1066.180,205.434,-83.899,173.085,29.918,155.468
C00825=1066.174,205.186,-83.876,173.082,29.916,155.467
C00826=1066.168,204.937,-83.851,173.081,29.912,155.467
C00827=1066.163,204.688,-83.827,173.078,29.909,155.466
C00828=1066.157,204.439,-83.802,173.075,29.906,155.466
C00829=1066.152,204.190,-83.778,173.074,29.903,155.465
C00830=1066.146,203.942,-83.754,173.071,29.899,155.465
C00831=1066.140,203.693,-83.730,173.069,29.896,155.464
C00832=1066.134,203.444,-83.705,173.067,29.893,155.464
C00833=1066.128,203.196,-83.680,173.065,29.890,155.463
C00834=1066.123,202.947,-83.656,173.062,29.887,155.463
C00835=1066.117,202.699,-83.632,173.061,29.884,155.462
C00836=1066.111,202.449,-83.608,173.058,29.880,155.462
C00837=1066.106,202.201,-83.583,173.056,29.877,155.461
C00838=1066.099,201.952,-83.559,173.054,29.874,155.461
C00839=1066.094,201.703,-83.535,173.052,29.871,155.460
C00840=1066.088,201.455,-83.511,173.049,29.868,155.460
C00841=1066.082,201.206,-83.487,173.048,29.865,155.459
C00842=1066.077,200.957,-83.463,173.045,29.862,155.459
C00843=1066.070,200.708,-83.439,173.042,29.858,155.458
C00844=1066.065,200.459,-83.415,173.041,29.855,155.458
C00845=1066.059,200.211,-83.391,173.038,29.852,155.457
C00846=1066.053,199.961,-83.367,173.036,29.849,155.457
C00847=1066.047,199.713,-83.343,173.034,29.846,155.457
C00848=1066.041,199.464,-83.318,173.032,29.843,155.456
C00849=1066.035,199.216,-83.295,173.029,29.840,155.456
C00850=1066.030,198.967,-83.270,173.028,29.837,155.455
C00851=1066.023,198.717,-83.247,173.025,29.834,155.455
C00852=1066.018,198.469,-83.223,173.023,29.831,155.454
C00853=1066.012,198.221,-83.199,173.021,29.828,155.454
C00854=1066.005,197.972,-83.175,173.019,29.825,155.453
C00855=1066.000,197.723,-83.151,173.016,29.821,155.453
C00856=1065.994,197.475,-83.127,173.015,29.819,155.452
C00857=1065.988,197.225,-83.103,173.012,29.815,155.452
C00858=1065.982,196.977,-83.080,173.010,29.813,155.451
C00859=1065.977,196.728,-83.055,173.008,29.809,155.451
C00860=1065.970,196.479,-83.031,173.006,29.806,155.450
C00861=1065.965,196.230,-83.008,173.003,29.803,155.450
C00862=1065.959,195.981,-82.984,173.002,29.800,155.449
C00863=1065.954,195.732,-82.960,172.999,29.797,155.449
C00864=1065.948,195.483,-82.937,172.997,29.794,155.448
C00865=1065.943,195.235,-82.912,172.996,29.791,155.448
C00866=1065.936,194.986,-82.889,172.993,29.788,155.448
C00867=1065.930,194.737,-82.865,172.991,29.785,155.447
C00868=1065.925,194.488,-82.841,172.989,29.782,155.447
C00869=1065.919,194.240,-82.818,172.987,29.778,155.446
C00870=1065.914,193.991,-82.794,172.984,29.776,155.446
C00871=1065.907,193.742,-82.770,172.983,29.772,155.445
C00872=1065.902,193.493,-82.746,172.980,29.769,155.445
C00873=1065.896,193.244,-82.723,172.978,29.766,155.444
C00874=1065.890,192.996,-82.699,172.976,29.763,155.444
C00875=1065.885,192.747,-82.676,172.974,29.760,155.443
C00876=1065.878,192.498,-82.652,172.972,29.757,155.443
C00877=1065.873,192.249,-82.627,172.970,29.754,155.442
C00878=1065.867,192.000,-82.604,172.968,29.751,155.442
C00879=1065.861,191.752,-82.581,172.965,29.748,155.441
C00880=1065.856,191.503,-82.557,172.964,29.745,155.441
C00881=1065.850,191.220,-82.530,172.961,29.741,155.440
C00882=1065.843,190.938,-82.503,172.959,29.738,155.440
C00883=1065.836,190.655,-82.476,172.957,29.735,155.439
C00884=1065.830,190.372,-82.450,172.954,29.731,155.439
C00885=1065.825,190.123,-82.426,172.952,29.728,155.438
C00886=1065.819,189.874,-82.403,172.950,29.725,155.438
C00887=1065.813,189.625,-82.378,172.948,29.722,155.437
C00888=1065.807,189.376,-82.355,172.946,29.719,155.437
C00889=1065.801,189.128,-82.332,172.944,29.716,155.436
C00890=1065.796,188.879,-82.308,172.941,29.712,155.436
C00891=1065.790,188.630,-82.285,172.940,29.710,155.436
C00892=1065.784,188.382,-82.262,172.937,29.706,155.435
C00893=1065.779,188.132,-82.238,172.935,29.704,155.435
C00894=1065.773,187.884,-82.214,172.934,29.700,155.434
C00895=1065.768,187.635,-82.192,172.931,29.697,155.434
C00896=1065.763,187.386,-82.168,172.929,29.694,155.433
C00897=1065.756,187.137,-82.144,172.927,29.691,155.433
C00898=1065.750,186.888,-82.121,172.925,29.688,155.432
C00899=1065.745,186.639,-82.097,172.923,29.685,155.432
C00900=1065.739,186.391,-82.074,172.921,29.682,155.431
C00901=1065.734,186.142,-82.051,172.919,29.679,155.431
C00902=1065.729,185.893,-82.027,172.917,29.676,155.430
C00903=1065.723,185.644,-82.004,172.915,29.673,155.430
C00904=1065.717,185.395,-81.981,172.913,29.670,155.429
C00905=1065.712,185.146,-81.957,172.911,29.666,155.429
C00906=1065.706,184.897,-81.934,172.909,29.664,155.428
C00907=1065.700,184.648,-81.911,172.907,29.661,155.428
C00908=1065.694,184.400,-81.888,172.905,29.658,155.428
C00909=1065.689,184.151,-81.865,172.903,29.655,155.427
C00910=1065.683,183.902,-81.842,172.901,29.652,155.427
C00911=1065.676,183.653,-81.818,172.899,29.649,155.426
C00912=1065.671,183.404,-81.795,172.897,29.646,155.426
C00913=1065.665,183.155,-81.773,172.894,29.643,155.425
C00914=1065.659,182.907,-81.749,172.893,29.640,155.425
C00915=1065.653,182.658,-81.726,172.891,29.637,155.424
C00916=1065.647,182.409,-81.704,172.888,29.635,155.424
C00917=1065.641,182.160,-81.681,172.886,29.632,155.424
C00918=1065.635,181.911,-81.658,172.885,29.629,155.423
C00919=1065.629,181.662,-81.634,172.882,29.626,155.423
C00920=1065.623,181.413,-81.611,172.880,29.623,155.422
C00921=1065.618,181.164,-81.588,172.878,29.620,155.422
C00922=1065.612,180.915,-81.566,172.876,29.617,155.421
C00923=1065.605,180.667,-81.543,172.874,29.614,155.421
C00924=1065.600,180.418,-81.520,172.872,29.611,155.421
C00925=1065.594,180.169,-81.497,172.870,29.609,155.420
C00926=1065.588,179.920,-81.474,172.868,29.605,155.420
C00927=1065.582,179.671,-81.451,172.866,29.603,155.419
C00928=1065.577,179.422,-81.428,172.864,29.600,155.419
C00929=1065.570,179.173,-81.406,172.862,29.597,155.418
C00930=1065.564,178.925,-81.383,172.860,29.594,155.418
C00931=1065.559,178.676,-81.360,172.858,29.591,155.418
C00932=1065.553,178.427,-81.337,172.856,29.588,155.417
C00933=1065.547,178.178,-81.314,172.854,29.585,155.417
C00934=1065.541,177.929,-81.292,172.852,29.582,155.416
C00935=1065.535,177.680,-81.269,172.850,29.580,155.416
C00936=1065.529,177.431,-81.246,172.848,29.577,155.415
C00937=1065.524,177.183,-81.223,172.846,29.573,155.415
C00938=1065.518,176.933,-81.201,172.844,29.571,155.414
C00939=1065.512,176.684,-81.178,172.842,29.568,155.414
C00940=1065.506,176.436,-81.156,172.840,29.565,155.414
C00941=1065.500,176.187,-81.133,172.839,29.562,155.413
C00942=1065.495,175.938,-81.110,172.836,29.559,155.413
C00943=1065.489,175.689,-81.087,172.834,29.556,155.412
C00944=1065.482,175.440,-81.064,172.833,29.553,155.412
C00945=1065.476,175.157,-81.039,172.830,29.550,155.411
C00946=1065.469,174.873,-81.013,172.828,29.547,155.411
C00947=1065.463,174.590,-80.987,172.826,29.543,155.410
C00948=1065.457,174.308,-80.961,172.823,29.540,155.410
C00949=1065.451,174.058,-80.939,172.821,29.537,155.409
C00950=1065.445,173.810,-80.917,172.820,29.534,155.409
C00951=1065.439,173.561,-80.894,172.817,29.531,155.409
C00952=1065.434,173.312,-80.871,172.815,29.528,155.408
C00953=1065.428,173.063,-80.849,172.814,29.526,155.408
C00954=1065.422,172.814,-80.826,172.812,29.523,155.407
C00955=1065.416,172.565,-80.803,172.809,29.520,155.407
C00956=1065.410,172.316,-80.780,172.808,29.517,155.406
C00957=1065.405,172.067,-80.759,172.806,29.514,155.406
C00958=1065.399,171.819,-80.736,172.803,29.511,155.405
C00959=1065.393,171.570,-80.713,172.802,29.508,155.405
C00960=1065.388,171.320,-80.691,172.800,29.505,155.405
C00961=1065.382,171.071,-80.668,172.798,29.502,155.404
C00962=1065.376,170.823,-80.646,172.796,29.499,155.404
C00963=1065.370,170.573,-80.624,172.794,29.497,155.403
C00964=1065.365,170.325,-80.601,172.792,29.494,155.403
C00965=1065.359,170.076,-80.579,172.791,29.491,155.402
C00966=1065.353,169.827,-80.556,172.788,29.488,155.402
C00967=1065.347,169.578,-80.533,172.787,29.485,155.402
C00968=1065.342,169.329,-80.511,172.785,29.482,155.401
C00969=1065.336,169.081,-80.489,172.783,29.479,155.401
C00970=1065.331,168.831,-80.467,172.781,29.476,155.400
C00971=1065.325,168.582,-80.444,172.779,29.473,155.400
C00972=1065.319,168.333,-80.422,172.777,29.470,155.399
C00973=1065.313,168.084,-80.399,172.776,29.468,155.399
C00974=1065.308,167.835,-80.378,172.773,29.465,155.398
C00975=1065.302,167.587,-80.355,172.771,29.461,155.398
C00976=1065.296,167.337,-80.333,172.770,29.459,155.398
C00977=1065.291,167.088,-80.310,172.768,29.456,155.397
C00978=1065.286,166.840,-80.288,172.765,29.453,155.397
C00979=1065.279,166.591,-80.266,172.764,29.450,155.396
C00980=1065.274,166.342,-80.244,172.762,29.447,155.396
C00981=1065.268,166.093,-80.221,172.760,29.444,155.395
C00982=1065.263,165.844,-80.199,172.758,29.441,155.395
C00983=1065.257,165.595,-80.176,172.756,29.438,155.394
C00984=1065.251,165.346,-80.154,172.754,29.435,155.394
C00985=1065.246,165.097,-80.133,172.753,29.432,155.394
C00986=1065.240,164.848,-80.110,172.751,29.430,155.393
C00987=1065.235,164.599,-80.088,172.748,29.427,155.393
C00988=1065.229,164.351,-80.066,172.747,29.423,155.392
C00989=1065.223,164.101,-80.044,172.745,29.421,155.392
C00990=1065.218,163.852,-80.021,172.743,29.418,155.391
C00991=1065.212,163.604,-79.999,172.741,29.415,155.391
C00992=1065.207,163.354,-79.977,172.739,29.412,155.390
C00993=1065.200,163.105,-79.955,172.738,29.409,155.390
C00994=1065.195,162.857,-79.933,172.736,29.406,155.390
C00995=1065.190,162.608,-79.911,172.734,29.403,155.389
C00996=1065.184,162.358,-79.889,172.732,29.400,155.389
C00997=1065.179,162.110,-79.866,172.730,29.397,155.388
C00998=1065.173,161.861,-79.844,172.728,29.394,155.388
C00999=1065.167,161.611,-79.823,172.727,29.392,155.387
C01000=1065.162,161.363,-79.800,172.725,29.388,155.387
C01001=1065.156,161.114,-79.778,172.723,29.386,155.386
C01002=1065.150,160.864,-79.756,172.721,29.383,155.386
C01003=1065.145,160.616,-79.735,172.719,29.380,155.386
C01004=1065.139,160.367,-79.713,172.717,29.377,155.385
C01005=1065.133,160.118,-79.690,172.716,29.374,155.385
C01006=1065.127,159.869,-79.669,172.714,29.371,155.384
C01007=1065.121,159.620,-79.647,172.711,29.368,155.384
C01008=1065.116,159.371,-79.625,172.710,29.366,155.383
C01009=1065.109,159.087,-79.600,172.708,29.363,155.383
C01010=1065.102,158.805,-79.576,172.706,29.360,155.383
C01011=1065.096,158.521,-79.551,172.704,29.356,155.382
C01012=1065.089,158.237,-79.526,172.701,29.353,155.382
C01013=1065.083,157.988,-79.504,172.700,29.350,155.381
C01014=1065.078,157.739,-79.483,172.698,29.347,155.381
C01015=1065.072,157.490,-79.461,172.696,29.345,155.380
C01016=1065.066,157.241,-79.439,172.694,29.342,155.380
C01017=1065.061,156.992,-79.417,172.692,29.339,155.379
C01018=1065.055,156.743,-79.396,172.690,29.336,155.379
C01019=1065.049,156.494,-79.374,172.689,29.333,155.379
C01020=1065.043,156.245,-79.353,172.687,29.330,155.378
C01021=1065.038,155.996,-79.331,172.685,29.328,155.378
C01022=1065.032,155.747,-79.309,172.683,29.325,155.377
C01023=1065.026,155.498,-79.288,172.681,29.322,155.377
C01024=1065.020,155.249,-79.266,172.680,29.319,155.376
C01025=1065.014,155.000,-79.245,172.678,29.316,155.376
C01026=1065.009,154.751,-79.223,172.676,29.313,155.376
C01027=1065.003,154.502,-79.201,172.675,29.311,155.375
C01028=1064.997,154.253,-79.180,172.672,29.308,155.375
C01029=1064.991,154.004,-79.158,172.670,29.305,155.374
C01030=1064.985,153.755,-79.137,172.669,29.302,155.374
C01031=1064.979,153.506,-79.115,172.667,29.300,155.374
C01032=1064.973,153.258,-79.094,172.665,29.296,155.373
C01033=1064.968,153.008,-79.072,172.664,29.294,155.373
C01034=1064.962,152.759,-79.050,172.662,29.291,155.372
C01035=1064.956,152.510,-79.029,172.659,29.288,155.372
C01036=1064.950,152.261,-79.007,172.658,29.285,155.371
C01037=1064.945,152.012,-78.987,172.656,29.283,155.371
C01038=1064.939,151.763,-78.965,172.654,29.280,155.371
C01039=1064.933,151.514,-78.944,172.653,29.277,155.370
C01040=1064.927,151.265,-78.922,172.651,29.274,155.370
C01041=1064.922,151.016,-78.900,172.649,29.271,155.369
C01042=1064.916,150.767,-78.879,172.647,29.268,155.369
C01043=1064.910,150.517,-78.858,172.645,29.266,155.369
C01044=1064.905,150.269,-78.836,172.643,29.263,155.368
C01045=1064.898,150.020,-78.815,172.642,29.260,155.368
C01046=1064.893,149.771,-78.793,172.640,29.257,155.367
C01047=1064.887,149.522,-78.772,172.638,29.255,155.367
C01048=1064.881,149.273,-78.751,172.637,29.251,155.366
C01049=1064.875,149.024,-78.730,172.635,29.249,155.366
C01050=1064.870,148.775,-78.708,172.633,29.246,155.366
C01051=1064.864,148.526,-78.687,172.631,29.243,155.365
C01052=1064.858,148.277,-78.666,172.629,29.240,155.365
C01053=1064.852,148.028,-78.645,172.628,29.238,155.364
C01054=1064.847,147.779,-78.623,172.626,29.235,155.364
C01055=1064.841,147.529,-78.602,172.624,29.232,155.364
C01056=1064.835,147.281,-78.581,172.623,29.230,155.363
C01057=1064.829,147.031,-78.559,172.621,29.227,155.363
C01058=1064.823,146.783,-78.538,172.618,29.224,155.362
C01059=1064.817,146.533,-78.518,172.617,29.221,155.362
C01060=1064.811,146.285,-78.497,172.615,29.218,155.361
C01061=1064.805,146.035,-78.476,172.613,29.215,155.361
C01062=1064.800,145.787,-78.454,172.612,29.212,155.361
C01063=1064.794,145.537,-78.433,172.610,29.210,155.360
C01064=1064.788,145.288,-78.412,172.608,29.207,155.360
C01065=1064.782,145.039,-78.391,172.607,29.204,155.359
C01066=1064.777,144.790,-78.370,172.605,29.202,155.359
C01067=1064.770,144.541,-78.349,172.603,29.199,155.359
C01068=1064.765,144.293,-78.328,172.601,29.196,155.358
C01069=1064.759,144.043,-78.307,172.599,29.193,155.358
C01070=1064.753,143.794,-78.285,172.598,29.191,155.357
C01071=1064.748,143.545,-78.265,172.596,29.188,155.357
C01072=1064.742,143.296,-78.243,172.594,29.185,155.357
C01073=1064.735,143.012,-78.219,172.593,29.182,155.356
C01074=1064.729,142.729,-78.196,172.590,29.178,155.355
C01075=1064.722,142.444,-78.172,172.588,29.176,155.355
C01076=1064.715,142.160,-78.148,172.587,29.172,155.355
C01077=1064.709,141.912,-78.127,172.584,29.169,155.354
C01078=1064.704,141.663,-78.106,172.583,29.167,155.354
C01079=1064.698,141.414,-78.085,172.581,29.164,155.353
C01080=1064.692,141.165,-78.064,172.579,29.161,155.353
C01081=1064.687,140.915,-78.043,172.578,29.159,155.353
C01082=1064.680,140.667,-78.023,172.576,29.156,155.352
C01083=1064.675,140.418,-78.002,172.574,29.153,155.352
C01084=1064.669,140.168,-77.980,172.573,29.150,155.351
C01085=1064.664,139.919,-77.960,172.571,29.147,155.351
C01086=1064.658,139.670,-77.938,172.569,29.144,155.350
C01087=1064.652,139.421,-77.918,172.568,29.142,155.350
C01088=1064.646,139.172,-77.898,172.566,29.139,155.350
C01089=1064.640,138.923,-77.876,172.565,29.136,155.349
C01090=1064.634,138.674,-77.856,172.562,29.133,155.349
C01091=1064.629,138.425,-77.836,172.560,29.131,155.348
C01092=1064.623,138.176,-77.814,172.559,29.128,155.348
C01093=1064.617,137.927,-77.794,172.557,29.125,155.348
C01094=1064.611,137.677,-77.773,172.555,29.122,155.347
C01095=1064.605,137.429,-77.752,172.554,29.120,155.347
C01096=1064.599,137.180,-77.732,172.552,29.117,155.346
C01097=1064.593,136.930,-77.711,172.550,29.114,155.346
C01098=1064.587,136.682,-77.690,172.549,29.111,155.346
C01099=1064.582,136.433,-77.670,172.547,29.109,155.345
C01100=1064.576,136.183,-77.649,172.545,29.106,155.345
C01101=1064.570,135.934,-77.629,172.544,29.103,155.344
C01102=1064.564,135.686,-77.608,172.542,29.101,155.344
C01103=1064.558,135.436,-77.587,172.540,29.098,155.343
C01104=1064.553,135.187,-77.567,172.539,29.095,155.343
C01105=1064.547,134.938,-77.546,172.537,29.092,155.343
C01106=1064.541,134.688,-77.526,172.536,29.090,155.342
C01107=1064.535,134.440,-77.505,172.534,29.087,155.342
C01108=1064.529,134.191,-77.485,172.531,29.084,155.341
C01109=1064.523,133.941,-77.464,172.530,29.081,155.341
C01110=1064.518,133.692,-77.443,172.528,29.079,155.341
C01111=1064.512,133.443,-77.423,172.526,29.076,155.340
C01112=1064.507,133.195,-77.402,172.525,29.073,155.340
C01113=1064.500,132.945,-77.382,172.523,29.070,155.339
C01114=1064.495,132.696,-77.361,172.521,29.067,155.339
C01115=1064.489,132.447,-77.341,172.520,29.064,155.339
C01116=1064.483,132.198,-77.320,172.518,29.062,155.338
C01117=1064.478,131.948,-77.300,172.517,29.059,155.338
C01118=1064.472,131.699,-77.280,172.515,29.056,155.337
C01119=1064.466,131.451,-77.260,172.513,29.053,155.337
C01120=1064.460,131.201,-77.239,172.512,29.051,155.336
C01121=1064.453,130.953,-77.218,172.510,29.048,155.336
C01122=1064.447,130.704,-77.198,172.508,29.046,155.336
C01123=1064.442,130.454,-77.177,172.507,29.043,155.335
C01124=1064.436,130.205,-77.157,172.505,29.040,155.335
C01125=1064.430,129.956,-77.137,172.503,29.038,155.335
C01126=1064.424,129.707,-77.117,172.502,29.035,155.334
C01127=1064.418,129.458,-77.096,172.500,29.032,155.334
C01128=1064.412,129.209,-77.076,172.498,29.029,155.333
C01129=1064.406,128.960,-77.056,172.497,29.027,155.333
C01130=1064.400,128.710,-77.036,172.495,29.024,155.333
C01131=1064.394,128.461,-77.016,172.493,29.021,155.332
C01132=1064.388,128.213,-76.996,172.492,29.019,155.332
C01133=1064.383,127.964,-76.975,172.490,29.016,155.331
C01134=1064.376,127.713,-76.955,172.489,29.013,155.331
C01135=1064.370,127.465,-76.936,172.487,29.010,155.331
C01136=1064.365,127.215,-76.915,172.485,29.008,155.330
C01137=1064.358,126.932,-76.892,172.483,29.005,155.330
C01138=1064.351,126.648,-76.869,172.481,29.001,155.329
C01139=1064.345,126.363,-76.846,172.479,28.999,155.329
C01140=1064.338,126.080,-76.823,172.477,28.995,155.328
C01141=1064.332,125.832,-76.803,172.475,28.992,155.328
C01142=1064.326,125.581,-76.783,172.474,28.990,155.328
C01143=1064.320,125.332,-76.763,172.472,28.987,155.327
C01144=1064.314,125.083,-76.743,172.470,28.984,155.327
C01145=1064.308,124.835,-76.723,172.469,28.981,155.326
C01146=1064.302,124.586,-76.703,172.467,28.979,155.326
C01147=1064.296,124.336,-76.682,172.465,28.976,155.325
C01148=1064.290,124.087,-76.662,172.464,28.973,155.325
C01149=1064.285,123.838,-76.643,172.462,28.970,155.325
C01150=1064.279,123.589,-76.623,172.460,28.968,155.324
C01151=1064.274,123.340,-76.602,172.459,28.966,155.324
C01152=1064.268,123.091,-76.582,172.457,28.963,155.324
C01153=1064.262,122.842,-76.562,172.456,28.960,155.323
C01154=1064.255,122.592,-76.543,172.454,28.957,155.323
C01155=1064.250,122.343,-76.522,172.453,28.955,155.322
C01156=1064.244,122.094,-76.502,172.452,28.952,155.322
C01157=1064.238,121.845,-76.482,172.450,28.949,155.322
C01158=1064.232,121.596,-76.463,172.448,28.946,155.321
C01159=1064.227,121.347,-76.442,172.447,28.943,155.321
C01160=1064.221,121.098,-76.423,172.445,28.941,155.320
C01161=1064.215,120.849,-76.403,172.444,28.938,155.320
C01162=1064.209,120.599,-76.383,172.442,28.935,155.319
C01163=1064.203,120.350,-76.363,172.440,28.932,155.319
C01164=1064.198,120.100,-76.343,172.439,28.930,155.319
C01165=1064.192,119.852,-76.323,172.437,28.927,155.318
C01166=1064.186,119.603,-76.303,172.435,28.924,155.318
C01167=1064.180,119.353,-76.284,172.434,28.921,155.317
C01168=1064.174,119.105,-76.264,172.432,28.919,155.317
C01169=1064.169,118.855,-76.243,172.430,28.916,155.317
C01170=1064.163,118.606,-76.224,172.429,28.913,155.316
C01171=1064.157,118.357,-76.204,172.427,28.910,155.316
C01172=1064.151,118.108,-76.184,172.426,28.908,155.315
C01173=1064.146,117.859,-76.165,172.424,28.905,155.315
C01174=1064.140,117.610,-76.145,172.422,28.902,155.315
C01175=1064.135,117.360,-76.125,172.421,28.899,155.314
C01176=1064.129,117.112,-76.105,172.419,28.897,155.314
C01177=1064.122,116.862,-76.085,172.417,28.894,155.313
C01178=1064.116,116.613,-76.066,172.416,28.891,155.313
C01179=1064.110,116.364,-76.046,172.414,28.889,155.312
C01180=1064.105,116.114,-76.026,172.413,28.886,155.312
C01181=1064.099,115.865,-76.006,172.411,28.883,155.312
C01182=1064.094,115.616,-75.987,172.409,28.880,155.311
C01183=1064.088,115.367,-75.967,172.408,28.877,155.311
C01184=1064.082,115.118,-75.948,172.406,28.874,155.310
C01185=1064.076,114.869,-75.928,172.404,28.871,155.310
C01186=1064.071,114.619,-75.908,172.404,28.869,155.310
C01187=1064.065,114.370,-75.888,172.402,28.866,155.309
C01188=1064.059,114.121,-75.869,172.401,28.863,155.309
C01189=1064.053,113.872,-75.849,172.399,28.861,155.308
C01190=1064.048,113.623,-75.829,172.397,28.858,155.308
C01191=1064.042,113.374,-75.809,172.396,28.855,155.307
C01192=1064.036,113.124,-75.790,172.394,28.852,155.307
C01193=1064.030,112.875,-75.771,172.392,28.850,155.307
C01194=1064.024,112.626,-75.751,172.391,28.847,155.306
C01195=1064.018,112.377,-75.732,172.389,28.844,155.306
C01196=1064.012,112.128,-75.712,172.388,28.842,155.305
C01197=1064.006,111.879,-75.693,172.386,28.839,155.305
C01198=1064.001,111.629,-75.674,172.384,28.836,155.305
C01199=1063.995,111.380,-75.654,172.383,28.833,155.304
C01200=1063.989,111.131,-75.635,172.381,28.831,155.304
C01201=1063.982,110.847,-75.612,172.379,28.828,155.303
C01202=1063.976,110.564,-75.590,172.378,28.825,155.303
C01203=1063.968,110.279,-75.569,172.376,28.822,155.303
C01204=1063.962,109.995,-75.546,172.374,28.819,155.302
C01205=1063.956,109.746,-75.527,172.372,28.816,155.302
C01206=1063.950,109.497,-75.508,172.370,28.813,155.301
C01207=1063.944,109.248,-75.488,172.370,28.811,155.301
C01208=1063.938,108.999,-75.469,172.368,28.808,155.301
C01209=1063.932,108.749,-75.450,172.366,28.805,155.300
C01210=1063.926,108.500,-75.430,172.365,28.802,155.300
C01211=1063.920,108.251,-75.411,172.363,28.800,155.299
C01212=1063.915,108.001,-75.391,172.362,28.797,155.299
C01213=1063.908,107.752,-75.373,172.360,28.794,155.299
C01214=1063.903,107.503,-75.354,172.358,28.791,155.298
C01215=1063.897,107.254,-75.334,172.357,28.789,155.298
C01216=1063.892,107.005,-75.315,172.355,28.786,155.297
C01217=1063.885,106.756,-75.296,172.354,28.783,155.297
C01218=1063.879,106.507,-75.277,172.352,28.780,155.297
C01219=1063.874,106.257,-75.258,172.350,28.778,155.296
C01220=1063.868,106.009,-75.238,172.349,28.776,155.296
C01221=1063.861,105.759,-75.219,172.347,28.773,155.295
C01222=1063.856,105.510,-75.200,172.346,28.770,155.295
C01223=1063.850,105.261,-75.181,172.345,28.768,155.295
C01224=1063.844,105.011,-75.161,172.343,28.765,155.294
C01225=1063.838,104.762,-75.143,172.341,28.762,155.294
C01226=1063.832,104.513,-75.123,172.340,28.759,155.293
C01227=1063.826,104.264,-75.103,172.338,28.757,155.293
C01228=1063.821,104.015,-75.085,172.337,28.754,155.293
C01229=1063.815,103.766,-75.066,172.335,28.751,155.292
C01230=1063.809,103.517,-75.047,172.333,28.748,155.292
C01231=1063.803,103.267,-75.027,172.332,28.745,155.291
C01232=1063.798,103.018,-75.008,172.330,28.743,155.291
C01233=1063.791,102.769,-74.990,172.329,28.740,155.291
C01234=1063.786,102.519,-74.970,172.327,28.737,155.290
C01235=1063.780,102.270,-74.951,172.326,28.735,155.290
C01236=1063.775,102.021,-74.932,172.325,28.732,155.289
C01237=1063.768,101.772,-74.914,172.323,28.729,155.289
C01238=1063.763,101.522,-74.894,172.321,28.726,155.289
C01239=1063.757,101.274,-74.874,172.320,28.724,155.288
C01240=1063.750,101.024,-74.856,172.318,28.721,155.288
C01241=1063.745,100.776,-74.837,172.317,28.718,155.287
C01242=1063.739,100.526,-74.819,172.315,28.715,155.287
C01243=1063.733,100.277,-74.800,172.313,28.713,155.287
C01244=1063.727,100.027,-74.781,172.312,28.710,155.286
C01245=1063.721,99.778,-74.762,172.310,28.707,155.286
C01246=1063.715,99.529,-74.743,172.309,28.705,155.285
C01247=1063.709,99.279,-74.724,172.308,28.702,155.285
C01248=1063.703,99.030,-74.705,172.306,28.700,155.285
C01249=1063.698,98.782,-74.686,172.305,28.697,155.284
C01250=1063.691,98.532,-74.668,172.303,28.694,155.284
C01251=1063.685,98.283,-74.648,172.301,28.691,155.283
C01252=1063.679,98.034,-74.630,172.300,28.689,155.283
C01253=1063.673,97.784,-74.611,172.298,28.686,155.283
C01254=1063.667,97.535,-74.592,172.297,28.683,155.282
C01255=1063.662,97.286,-74.574,172.295,28.680,155.282
C01256=1063.656,97.037,-74.555,172.293,28.678,155.281
C01257=1063.650,96.787,-74.536,172.293,28.675,155.281
C01258=1063.644,96.538,-74.517,172.291,28.673,155.281
C01259=1063.638,96.289,-74.498,172.289,28.670,155.280
C01260=1063.632,96.040,-74.480,172.288,28.667,155.280
C01261=1063.626,95.791,-74.460,172.286,28.665,155.279
C01262=1063.620,95.541,-74.442,172.285,28.662,155.279
C01263=1063.615,95.292,-74.423,172.283,28.659,155.279
C01264=1063.608,95.043,-74.405,172.281,28.656,155.278
C01265=1063.600,94.676,-74.377,172.279,28.652,155.278
C01266=1063.591,94.310,-74.350,172.277,28.648,155.277
C01267=1063.582,93.943,-74.322,172.275,28.644,155.276
C01268=1063.574,93.577,-74.295,172.273,28.641,155.276
C01269=1063.568,93.328,-74.277,172.271,28.638,155.276
C01270=1063.563,93.079,-74.257,172.269,28.635,155.275
C01271=1063.556,92.830,-74.239,172.268,28.632,155.275
C01272=1063.550,92.580,-74.221,172.267,28.630,155.274
C01273=1063.545,92.331,-74.202,172.265,28.627,155.274
C01274=1063.539,92.082,-74.183,172.264,28.624,155.273
C01275=1063.533,91.833,-74.164,172.262,28.621,155.273
C01276=1063.527,91.584,-74.146,172.261,28.619,155.273
C01277=1063.522,91.334,-74.127,172.259,28.616,155.272
C01278=1063.515,91.085,-74.109,172.257,28.613,155.272
C01279=1063.509,90.835,-74.091,172.256,28.610,155.271
C01280=1063.504,90.587,-74.072,172.254,28.608,155.271
C01281=1063.498,90.337,-74.054,172.254,28.605,155.271
C01282=1063.492,90.088,-74.035,172.252,28.602,155.270
C01283=1063.485,89.839,-74.017,172.250,28.600,155.270
C01284=1063.480,89.589,-73.998,172.249,28.597,155.270
C01285=1063.474,89.340,-73.980,172.247,28.595,155.269
C01286=1063.468,89.090,-73.962,172.245,28.592,155.269
C01287=1063.461,88.841,-73.943,172.244,28.589,155.268
C01288=1063.456,88.593,-73.925,172.242,28.586,155.268
C01289=1063.450,88.343,-73.906,172.241,28.584,155.268
C01290=1063.444,88.094,-73.888,172.240,28.582,155.267
C01291=1063.438,87.845,-73.870,172.238,28.579,155.267
C01292=1063.432,87.596,-73.851,172.237,28.576,155.266
C01293=1063.426,87.346,-73.834,172.235,28.573,155.266
C01294=1063.419,87.097,-73.815,172.234,28.570,155.266
C01295=1063.414,86.847,-73.797,172.232,28.568,155.265
C01296=1063.408,86.598,-73.778,172.230,28.565,155.265
C01297=1063.402,86.348,-73.760,172.229,28.562,155.264
C01298=1063.396,86.100,-73.742,172.228,28.560,155.264
C01299=1063.390,85.850,-73.724,172.226,28.557,155.264
C01300=1063.384,85.601,-73.705,172.225,28.555,155.263
C01301=1063.379,85.352,-73.687,172.223,28.552,155.263
C01302=1063.372,85.103,-73.668,172.222,28.549,155.263
C01303=1063.366,84.853,-73.651,172.220,28.546,155.262
C01304=1063.360,84.605,-73.632,172.218,28.544,155.262
C01305=1063.354,84.355,-73.614,172.217,28.541,155.261
C01306=1063.348,84.106,-73.596,172.216,28.538,155.261
C01307=1063.343,83.856,-73.578,172.215,28.536,155.261
C01308=1063.337,83.607,-73.560,172.213,28.533,155.260
C01309=1063.327,83.191,-73.529,172.211,28.529,155.260
C01310=1063.317,82.775,-73.499,172.208,28.524,155.259
C01311=1063.307,82.359,-73.469,172.205,28.519,155.258
C01312=1063.297,81.943,-73.439,172.203,28.515,155.258
C01313=1063.291,81.693,-73.421,172.201,28.512,155.257
C01314=1063.285,81.445,-73.402,172.200,28.509,155.257
C01315=1063.279,81.195,-73.384,172.199,28.507,155.256
C01316=1063.274,80.945,-73.366,172.197,28.504,155.256
C01317=1063.268,80.697,-73.348,172.196,28.502,155.256
C01318=1063.262,80.447,-73.330,172.194,28.499,155.255
C01319=1063.257,80.198,-73.312,172.192,28.496,155.255
C01320=1063.250,79.948,-73.294,172.191,28.493,155.254
C01321=1063.245,79.700,-73.276,172.190,28.491,155.254
C01322=1063.238,79.450,-73.258,172.189,28.488,155.254
C01323=1063.233,79.201,-73.240,172.187,28.485,155.253
C01324=1063.227,78.952,-73.222,172.185,28.482,155.253
C01325=1063.220,78.667,-73.201,172.184,28.480,155.252
C01326=1063.213,78.384,-73.181,172.182,28.476,155.252
C01327=1063.207,78.100,-73.160,172.181,28.474,155.251
C01328=1063.200,77.816,-73.139,172.178,28.470,155.251
C01329=1063.194,77.567,-73.122,172.178,28.467,155.251
C01330=1063.188,77.317,-73.104,172.176,28.465,155.250
C01331=1063.182,77.068,-73.087,172.174,28.462,155.250
C01332=1063.176,76.818,-73.069,172.173,28.460,155.249
C01333=1063.170,76.570,-73.051,172.171,28.457,155.249
C01334=1063.164,76.320,-73.033,172.170,28.454,155.249
C01335=1063.158,76.070,-73.015,172.168,28.451,155.248
C01336=1063.152,75.821,-72.997,172.167,28.449,155.248
C01337=1063.146,75.572,-72.979,172.166,28.447,155.248
C01338=1063.141,75.323,-72.962,172.164,28.444,155.247
C01339=1063.134,75.073,-72.944,172.162,28.441,155.247
C01340=1063.128,74.825,-72.926,172.161,28.438,155.246
C01341=1063.122,74.575,-72.908,172.159,28.436,155.246
C01342=1063.116,74.326,-72.891,172.158,28.433,155.246
C01343=1063.110,74.076,-72.873,172.157,28.430,155.245
C01344=1063.105,73.827,-72.855,172.155,28.427,155.245
C01345=1063.098,73.577,-72.837,172.154,28.425,155.244
C01346=1063.093,73.328,-72.820,172.152,28.422,155.244
C01347=1063.086,73.079,-72.802,172.151,28.420,155.244
C01348=1063.081,72.830,-72.785,172.149,28.417,155.243
C01349=1063.074,72.580,-72.767,172.147,28.414,155.243
C01350=1063.069,72.331,-72.749,172.147,28.412,155.242
C01351=1063.063,72.081,-72.731,172.145,28.409,155.242
C01352=1063.057,71.832,-72.714,172.144,28.406,155.242
C01353=1063.050,71.583,-72.696,172.142,28.404,155.241
C01354=1063.045,71.334,-72.679,172.140,28.401,155.241
C01355=1063.039,71.084,-72.661,172.139,28.398,155.241
C01356=1063.033,70.835,-72.643,172.137,28.395,155.240
C01357=1063.027,70.585,-72.625,172.137,28.393,155.240
C01358=1063.021,70.337,-72.608,172.135,28.390,155.239
C01359=1063.015,70.088,-72.591,172.133,28.387,155.239
C01360=1063.009,69.838,-72.573,172.132,28.385,155.239
C01361=1063.004,69.589,-72.555,172.130,28.382,155.238
C01362=1062.998,69.339,-72.537,172.129,28.380,155.238
C01363=1062.991,69.090,-72.521,172.127,28.377,155.238
C01364=1062.985,68.841,-72.503,172.126,28.374,155.237
C01365=1062.980,68.592,-72.485,172.125,28.371,155.237
C01366=1062.973,68.342,-72.468,172.123,28.369,155.236
C01367=1062.967,68.093,-72.450,172.122,28.366,155.236
C01368=1062.962,67.843,-72.433,172.120,28.364,155.236
C01369=1062.955,67.594,-72.416,172.118,28.361,155.235
C01370=1062.950,67.345,-72.398,172.117,28.358,155.235
C01371=1062.944,67.095,-72.380,172.116,28.356,155.234
C01372=1062.937,66.847,-72.363,172.115,28.353,155.234
C01373=1062.931,66.597,-72.346,172.113,28.351,155.234
C01374=1062.926,66.348,-72.328,172.111,28.348,155.233
C01375=1062.920,66.098,-72.312,172.110,28.345,155.233
C01376=1062.914,65.849,-72.294,172.108,28.342,155.233
C01377=1062.908,65.600,-72.276,172.107,28.339,155.232
C01378=1062.901,65.350,-72.259,172.106,28.337,155.232
C01379=1062.896,65.101,-72.241,172.104,28.335,155.231
C01380=1062.890,64.852,-72.225,172.103,28.332,155.231
C01381=1062.884,64.602,-72.207,172.101,28.329,155.231
C01382=1062.878,64.353,-72.190,172.100,28.326,155.230
C01383=1062.871,64.104,-72.172,172.098,28.323,155.230
C01384=1062.866,63.854,-72.155,172.096,28.321,155.230
C01385=1062.860,63.605,-72.138,172.096,28.319,155.229
C01386=1062.853,63.356,-72.121,172.094,28.316,155.229
C01387=1062.848,63.107,-72.103,172.093,28.313,155.228
C01388=1062.841,62.857,-72.087,172.091,28.311,155.228
C01389=1062.834,62.573,-72.068,172.089,28.308,155.228
C01390=1062.827,62.289,-72.047,172.088,28.305,155.227
C01391=1062.821,62.005,-72.028,172.086,28.302,155.227
C01392=1062.813,61.721,-72.008,172.085,28.299,155.226
C01393=1062.807,61.471,-71.992,172.083,28.296,155.226
C01394=1062.801,61.222,-71.974,172.082,28.294,155.226
C01395=1062.795,60.973,-71.957,172.080,28.291,155.225
C01396=1062.788,60.723,-71.940,172.078,28.289,155.225
C01397=1062.783,60.474,-71.923,172.077,28.286,155.224
C01398=1062.777,60.225,-71.906,172.075,28.283,155.224
C01399=1062.771,59.975,-71.889,172.074,28.281,155.224
C01400=1062.765,59.726,-71.872,172.073,28.278,155.223
C01401=1062.759,59.477,-71.855,172.071,28.275,155.223
C01402=1062.752,59.227,-71.837,172.070,28.273,155.223
C01403=1062.746,58.978,-71.820,172.068,28.270,155.222
C01404=1062.740,58.729,-71.804,172.067,28.268,155.222
C01405=1062.734,58.479,-71.786,172.066,28.265,155.221
C01406=1062.728,58.230,-71.770,172.064,28.262,155.221
C01407=1062.722,57.981,-71.753,172.063,28.260,155.221
C01408=1062.716,57.731,-71.736,172.061,28.257,155.220
C01409=1062.710,57.482,-71.719,172.060,28.255,155.220
C01410=1062.705,57.232,-71.702,172.058,28.252,155.220
C01411=1062.698,56.983,-71.685,172.056,28.250,155.219
C01412=1062.692,56.734,-71.668,172.056,28.247,155.219
C01413=1062.686,56.484,-71.651,172.054,28.244,155.219
C01414=1062.679,56.235,-71.634,172.053,28.241,155.218
C01415=1062.673,55.986,-71.617,172.051,28.239,155.218
C01416=1062.668,55.737,-71.600,172.049,28.236,155.217
C01417=1062.662,55.487,-71.583,172.048,28.234,155.217
C01418=1062.655,55.237,-71.567,172.046,28.231,155.217
C01419=1062.650,54.988,-71.549,172.045,28.229,155.216
C01420=1062.644,54.739,-71.533,172.044,28.226,155.216
C01421=1062.637,54.489,-71.516,172.042,28.223,155.216
C01422=1062.632,54.240,-71.499,172.041,28.220,155.215
C01423=1062.626,53.991,-71.482,172.039,28.218,155.215
C01424=1062.620,53.742,-71.466,172.038,28.215,155.215
C01425=1062.613,53.492,-71.448,172.037,28.213,155.214
C01426=1062.608,53.243,-71.431,172.035,28.210,155.214
C01427=1062.602,52.993,-71.415,172.034,28.207,155.213
C01428=1062.595,52.744,-71.398,172.032,28.205,155.213
C01429=1062.590,52.495,-71.381,172.031,28.202,155.213
C01430=1062.583,52.245,-71.364,172.029,28.199,155.212
C01431=1062.577,51.996,-71.348,172.027,28.197,155.212
C01432=1062.572,51.746,-71.331,172.027,28.194,155.211
C01433=1062.566,51.498,-71.314,172.025,28.192,155.211
C01434=1062.559,51.248,-71.297,172.024,28.189,155.211
C01435=1062.553,50.998,-71.281,172.022,28.186,155.210
C01436=1062.548,50.749,-71.263,172.021,28.183,155.210
C01437=1062.542,50.500,-71.247,172.019,28.181,155.210
C01438=1062.536,50.250,-71.231,172.018,28.179,155.209
C01439=1062.531,50.001,-71.213,172.017,28.176,155.209
C01440=1062.524,49.751,-71.197,172.015,28.173,155.208
C01441=1062.518,49.502,-71.180,172.014,28.170,155.208
C01442=1062.512,49.253,-71.164,172.012,28.167,155.208
C01443=1062.507,49.004,-71.147,172.010,28.165,155.207
C01444=1062.501,48.754,-71.130,172.010,28.163,155.207
C01445=1062.495,48.505,-71.114,172.008,28.160,155.207
C01446=1062.488,48.255,-71.098,172.007,28.157,155.206
C01447=1062.483,48.006,-71.080,172.005,28.154,155.206
C01448=1062.477,47.757,-71.064,172.003,28.152,155.205
C01449=1062.471,47.507,-71.047,172.002,28.149,155.205
C01450=1062.465,47.258,-71.031,172.000,28.146,155.205
C01451=1062.459,47.009,-71.014,172.000,28.144,155.204
C01452=1062.453,46.759,-70.997,171.998,28.141,155.204
C01453=1062.446,46.475,-70.978,171.997,28.138,155.203
C01454=1062.440,46.190,-70.960,171.995,28.135,155.203
C01455=1062.433,45.906,-70.941,171.993,28.132,155.203
C01456=1062.426,45.621,-70.922,171.991,28.129,155.202
C01457=1062.420,45.373,-70.905,171.990,28.126,155.202
C01458=1062.415,45.123,-70.888,171.989,28.124,155.201
C01459=1062.409,44.874,-70.872,171.987,28.121,155.201
C01460=1062.403,44.624,-70.856,171.986,28.119,155.201
C01461=1062.397,44.375,-70.840,171.984,28.116,155.200
C01462=1062.391,44.125,-70.823,171.982,28.113,155.200
C01463=1062.386,43.876,-70.806,171.982,28.110,155.200
C01464=1062.379,43.627,-70.789,171.980,28.108,155.199
C01465=1062.373,43.377,-70.773,171.979,28.105,155.199
C01466=1062.367,43.128,-70.757,171.977,28.103,155.198
C01467=1062.361,42.878,-70.740,171.976,28.100,155.198
C01468=1062.355,42.629,-70.724,171.974,28.098,155.198
C01469=1062.349,42.380,-70.708,171.972,28.095,155.197
C01470=1062.343,42.130,-70.692,171.972,28.092,155.197
C01471=1062.337,41.881,-70.675,171.970,28.089,155.197
C01472=1062.331,41.632,-70.659,171.969,28.087,155.196
C01473=1062.325,41.382,-70.643,171.967,28.084,155.196
C01474=1062.319,41.133,-70.627,171.965,28.082,155.196
C01475=1062.313,40.884,-70.610,171.964,28.079,155.195
C01476=1062.307,40.633,-70.594,171.963,28.077,155.195
C01477=1062.301,40.384,-70.577,171.962,28.074,155.194
C01478=1062.295,40.135,-70.561,171.960,28.071,155.194
C01479=1062.289,39.885,-70.545,171.958,28.069,155.194
C01480=1062.283,39.636,-70.529,171.957,28.066,155.193
C01481=1062.277,39.387,-70.512,171.955,28.063,155.193
C01482=1062.271,39.137,-70.496,171.954,28.061,155.193
C01483=1062.265,38.888,-70.480,171.953,28.059,155.192
C01484=1062.259,38.639,-70.464,171.952,28.056,155.192
C01485=1062.253,38.389,-70.447,171.950,28.053,155.191
C01486=1062.247,38.140,-70.431,171.948,28.051,155.191
C01487=1062.241,37.891,-70.415,171.947,28.048,155.191
C01488=1062.236,37.641,-70.399,171.945,28.045,155.190
C01489=1062.230,37.391,-70.383,171.945,28.043,155.190
C01490=1062.223,37.142,-70.367,171.943,28.040,155.190
C01491=1062.217,36.893,-70.351,171.941,28.037,155.189
C01492=1062.211,36.644,-70.335,171.940,28.035,155.189
C01493=1062.205,36.394,-70.319,171.938,28.032,155.189
C01494=1062.199,36.145,-70.302,171.937,28.030,155.188
C01495=1062.193,35.895,-70.287,171.935,28.027,155.188
C01496=1062.186,35.645,-70.271,171.934,28.025,155.188
C01497=1062.180,35.396,-70.255,171.933,28.023,155.187
C01498=1062.174,35.147,-70.238,171.931,28.020,155.187
C01499=1062.168,34.897,-70.222,171.930,28.017,155.186
C01500=1062.162,34.648,-70.206,171.928,28.015,155.186
C01501=1062.156,34.398,-70.191,171.927,28.012,155.186
C01502=1062.150,34.149,-70.175,171.925,28.010,155.186
C01503=1062.144,33.899,-70.158,171.924,28.007,155.185
C01504=1062.137,33.650,-70.143,171.923,28.004,155.185
C01505=1062.132,33.400,-70.127,171.921,28.002,155.184
C01506=1062.126,33.151,-70.111,171.920,27.999,155.184
C01507=1062.120,32.902,-70.095,171.918,27.996,155.184
C01508=1062.114,32.652,-70.078,171.916,27.994,155.183
C01509=1062.108,32.403,-70.063,171.915,27.991,155.183
C01510=1062.102,32.153,-70.047,171.914,27.989,155.183
C01511=1062.096,31.905,-70.031,171.913,27.987,155.182
C01512=1062.090,31.655,-70.015,171.911,27.984,155.182
C01513=1062.084,31.406,-70.000,171.909,27.982,155.182
C01514=1062.078,31.156,-69.984,171.908,27.979,155.181
C01515=1062.072,30.907,-69.968,171.906,27.976,155.181
C01516=1062.066,30.657,-69.952,171.905,27.974,155.181
C01517=1062.059,30.373,-69.934,171.903,27.971,155.180
C01518=1062.052,30.089,-69.916,171.902,27.967,155.180
C01519=1062.045,29.804,-69.898,171.900,27.965,155.179
C01520=1062.038,29.520,-69.880,171.899,27.962,155.179
C01521=1062.032,29.270,-69.864,171.897,27.960,155.179
C01522=1062.026,29.021,-69.848,171.895,27.957,155.178
C01523=1062.020,28.771,-69.832,171.894,27.954,155.178
C01524=1062.014,28.522,-69.817,171.893,27.952,155.178
C01525=1062.009,28.273,-69.801,171.892,27.949,155.177
C01526=1062.002,28.023,-69.786,171.890,27.947,155.177
C01527=1061.996,27.774,-69.770,171.888,27.944,155.176
C01528=1061.991,27.524,-69.754,171.887,27.941,155.176
C01529=1061.984,27.275,-69.738,171.885,27.939,155.176
C01530=1061.978,27.026,-69.722,171.884,27.936,155.175
C01531=1061.972,26.776,-69.707,171.883,27.934,155.175
C01532=1061.966,26.527,-69.691,171.882,27.931,155.175
C01533=1061.960,26.277,-69.675,171.880,27.929,155.174
C01534=1061.953,26.028,-69.660,171.878,27.926,155.174
C01535=1061.948,25.778,-69.644,171.877,27.924,155.174
C01536=1061.942,25.529,-69.629,171.875,27.921,155.173
C01537=1061.936,25.279,-69.613,171.874,27.918,155.173
C01538=1061.929,25.030,-69.598,171.873,27.916,155.173
C01539=1061.924,24.780,-69.582,171.871,27.914,155.172
C01540=1061.917,24.531,-69.566,171.870,27.911,155.172
C01541=1061.911,24.281,-69.551,171.868,27.909,155.172
C01542=1061.905,24.032,-69.535,171.867,27.906,155.171
C01543=1061.899,23.782,-69.520,171.865,27.904,155.171
C01544=1061.892,23.533,-69.504,171.863,27.901,155.171
C01545=1061.887,23.284,-69.489,171.863,27.899,155.170
C01546=1061.881,23.034,-69.474,171.861,27.896,155.170
C01547=1061.875,22.785,-69.458,171.860,27.894,155.170
C01548=1061.868,22.535,-69.443,171.858,27.891,155.169
C01549=1061.862,22.286,-69.426,171.857,27.889,155.169
C01550=1061.856,22.036,-69.411,171.855,27.886,155.169
C01551=1061.851,21.787,-69.396,171.853,27.884,155.168
C01552=1061.844,21.538,-69.381,171.852,27.881,155.168
C01553=1061.839,21.288,-69.365,171.851,27.879,155.168
C01554=1061.832,21.039,-69.349,171.850,27.876,155.167
C01555=1061.826,20.789,-69.334,171.848,27.874,155.167
C01556=1061.820,20.539,-69.319,171.846,27.871,155.167
C01557=1061.815,20.291,-69.303,171.845,27.869,155.166
C01558=1061.808,20.041,-69.288,171.843,27.866,155.166
C01559=1061.803,19.791,-69.273,171.842,27.864,155.166
C01560=1061.796,19.542,-69.257,171.841,27.861,155.165
C01561=1061.790,19.292,-69.242,171.839,27.859,155.165
C01562=1061.784,19.043,-69.227,171.838,27.856,155.165
C01563=1061.778,18.794,-69.211,171.836,27.854,155.164
C01564=1061.771,18.544,-69.196,171.835,27.851,155.164
C01565=1061.766,18.294,-69.181,171.833,27.849,155.164
C01566=1061.759,18.045,-69.166,171.832,27.846,155.163
C01567=1061.754,17.796,-69.150,171.830,27.843,155.163
C01568=1061.748,17.547,-69.135,171.829,27.841,155.162
C01569=1061.741,17.297,-69.120,171.828,27.839,155.162
C01570=1061.736,17.047,-69.104,171.826,27.836,155.162
C01571=1061.729,16.798,-69.089,171.825,27.834,155.162
C01572=1061.723,16.549,-69.074,171.823,27.831,155.161
C01573=1061.718,16.299,-69.059,171.821,27.829,155.161
C01574=1061.711,16.049,-69.044,171.820,27.826,155.161
C01575=1061.705,15.800,-69.029,171.818,27.823,155.160
C01576=1061.699,15.551,-69.013,171.818,27.821,155.160
C01577=1061.693,15.301,-68.998,171.816,27.819,155.160
C01578=1061.687,15.052,-68.983,171.814,27.816,155.159
C01579=1061.681,14.802,-68.967,171.813,27.814,155.159
C01580=1061.675,14.553,-68.953,171.811,27.811,155.159
C01581=1061.668,14.270,-68.936,171.810,27.808,155.158
C01582=1061.661,13.987,-68.918,171.808,27.806,155.158
C01583=1061.654,13.704,-68.901,171.807,27.803,155.157
C01584=1061.647,13.420,-68.885,171.805,27.800,155.157
C01585=1061.641,13.171,-68.868,171.804,27.798,155.157
C01586=1061.634,12.921,-68.853,171.802,27.795,155.157
C01587=1061.629,12.672,-68.839,171.800,27.793,155.156
C01588=1061.622,12.423,-68.824,171.799,27.790,155.156
C01589=1061.616,12.173,-68.809,171.797,27.788,155.156
C01590=1061.609,11.923,-68.794,171.796,27.785,155.155
C01591=1061.604,11.675,-68.779,171.794,27.783,155.155
C01592=1061.597,11.425,-68.765,171.793,27.781,155.155
C01593=1061.592,11.175,-68.749,171.792,27.778,155.154
C01594=1061.585,10.925,-68.734,171.790,27.776,155.154
C01595=1061.579,10.676,-68.719,171.789,27.774,155.154
C01596=1061.573,10.427,-68.705,171.787,27.771,155.153
C01597=1061.567,10.177,-68.690,171.785,27.769,155.153
C01598=1061.561,9.928,-68.675,171.784,27.766,155.153
C01599=1061.555,9.678,-68.660,171.782,27.764,155.152
C01600=1061.548,9.429,-68.645,171.781,27.761,155.152
C01601=1061.542,9.179,-68.630,171.780,27.759,155.152
C01602=1061.536,8.930,-68.616,171.778,27.756,155.151
C01603=1061.530,8.680,-68.601,171.777,27.754,155.151
C01604=1061.524,8.430,-68.585,171.775,27.752,155.151
C01605=1061.518,8.182,-68.571,171.774,27.749,155.150
C01606=1061.512,7.932,-68.556,171.772,27.747,155.150
C01607=1061.505,7.682,-68.541,171.770,27.745,155.150
C01608=1061.500,7.433,-68.526,171.769,27.742,155.150
C01609=1061.493,7.184,-68.511,171.767,27.740,155.149
C01610=1061.487,6.934,-68.496,171.767,27.738,155.149
C01611=1061.481,6.685,-68.482,171.765,27.735,155.149
C01612=1061.475,6.435,-68.467,171.764,27.732,155.148
C01613=1061.469,6.185,-68.452,171.762,27.730,155.148
C01614=1061.463,5.936,-68.438,171.760,27.727,155.148
C01615=1061.456,5.686,-68.423,171.759,27.725,155.147
C01616=1061.451,5.437,-68.408,171.757,27.723,155.147
C01617=1061.444,5.188,-68.393,171.756,27.720,155.147
C01618=1061.438,4.938,-68.378,171.754,27.718,155.146
C01619=1061.433,4.689,-68.363,171.753,27.716,155.146
C01620=1061.427,4.439,-68.349,171.752,27.713,155.146
C01621=1061.420,4.189,-68.334,171.750,27.711,155.145
C01622=1061.415,3.940,-68.319,171.749,27.708,155.145
C01623=1061.408,3.690,-68.305,171.747,27.706,155.145
C01624=1061.402,3.441,-68.290,171.745,27.703,155.145
C01625=1061.396,3.191,-68.276,171.744,27.701,155.144
C01626=1061.391,2.942,-68.261,171.742,27.698,155.144
C01627=1061.384,2.692,-68.246,171.741,27.696,155.144
C01628=1061.378,2.443,-68.231,171.739,27.694,155.143
C01629=1061.372,2.194,-68.217,171.738,27.691,155.143
C01630=1061.366,1.944,-68.202,171.737,27.689,155.143
C01631=1061.360,1.695,-68.188,171.735,27.687,155.142
C01632=1061.354,1.445,-68.173,171.734,27.684,155.142
C01633=1061.348,1.196,-68.158,171.732,27.682,155.142
C01634=1061.342,0.946,-68.144,171.731,27.679,155.141
C01635=1061.336,0.697,-68.129,171.729,27.676,155.141
C01636=1061.330,0.447,-68.115,171.727,27.674,155.141
C01637=1061.324,0.197,-68.100,171.726,27.672,155.141
C01638=1061.318,-0.052,-68.086,171.724,27.670,155.140
C01639=1061.312,-0.302,-68.071,171.724,27.667,155.140
C01640=1061.306,-0.551,-68.057,171.722,27.665,155.140
C01641=1061.300,-0.801,-68.042,171.720,27.663,155.139
C01642=1061.294,-1.050,-68.027,171.719,27.660,155.139
C01643=1061.288,-1.300,-68.013,171.717,27.657,155.139
C01644=1061.282,-1.549,-67.999,171.716,27.655,155.138
C01645=1061.275,-1.830,-67.982,171.714,27.652,155.138
C01646=1061.269,-2.111,-67.966,171.713,27.650,155.138
C01647=1061.262,-2.392,-67.950,171.711,27.647,155.137
C01648=1061.255,-2.673,-67.933,171.709,27.644,155.137
C01649=1061.249,-2.923,-67.919,171.708,27.642,155.137
C01650=1061.243,-3.172,-67.904,171.706,27.639,155.136
C01651=1061.237,-3.422,-67.890,171.705,27.637,155.136
C01652=1061.231,-3.671,-67.876,171.703,27.635,155.136
C01653=1061.225,-3.921,-67.862,171.702,27.633,155.135
C01654=1061.219,-4.170,-67.847,171.700,27.630,155.135
C01655=1061.212,-4.420,-67.833,171.698,27.627,155.135
C01656=1061.206,-4.670,-67.819,171.697,27.625,155.135
C01657=1061.200,-4.919,-67.804,171.695,27.623,155.134
C01658=1061.194,-5.169,-67.790,171.694,27.621,155.134
C01659=1061.187,-5.418,-67.776,171.692,27.618,155.134
C01660=1061.181,-5.668,-67.762,171.691,27.616,155.133
C01661=1061.175,-5.917,-67.747,171.690,27.614,155.133
C01662=1061.169,-6.167,-67.733,171.688,27.612,155.133
C01663=1061.163,-6.416,-67.719,171.687,27.609,155.133
C01664=1061.157,-6.666,-67.705,171.685,27.607,155.132
C01665=1061.150,-6.915,-67.691,171.683,27.604,155.132
C01666=1061.144,-7.165,-67.676,171.682,27.602,155.132
C01667=1061.139,-7.415,-67.662,171.680,27.600,155.131
C01668=1061.133,-7.664,-67.648,171.679,27.598,155.131
C01669=1061.126,-7.914,-67.634,171.677,27.595,155.131
C01670=1061.120,-8.163,-67.620,171.675,27.593,155.131
C01671=1061.114,-8.413,-67.605,171.674,27.590,155.130
C01672=1061.108,-8.662,-67.591,171.672,27.588,155.130
C01673=1061.102,-8.912,-67.577,171.672,27.586,155.130
C01674=1061.096,-9.161,-67.563,171.670,27.584,155.129
C01675=1061.089,-9.411,-67.549,171.668,27.582,155.129
C01676=1061.084,-9.660,-67.535,171.667,27.579,155.129
C01677=1061.078,-9.909,-67.521,171.665,27.577,155.129
C01678=1061.071,-10.159,-67.507,171.663,27.575,155.128
C01679=1061.065,-10.409,-67.493,171.662,27.572,155.128
C01680=1061.058,-10.658,-67.479,171.660,27.570,155.128
C01681=1061.053,-10.908,-67.465,171.659,27.567,155.127
C01682=1061.047,-11.157,-67.451,171.657,27.565,155.127
C01683=1061.040,-11.407,-67.437,171.656,27.563,155.127
C01684=1061.035,-11.656,-67.423,171.654,27.561,155.127
C01685=1061.029,-11.907,-67.409,171.652,27.558,155.126
C01686=1061.022,-12.155,-67.395,171.651,27.556,155.126
C01687=1061.017,-12.405,-67.381,171.650,27.554,155.126
C01688=1061.011,-12.655,-67.366,171.648,27.552,155.125
C01689=1061.004,-12.904,-67.352,171.647,27.549,155.125
C01690=1060.999,-13.153,-67.339,171.645,27.547,155.125
C01691=1060.992,-13.403,-67.325,171.644,27.545,155.125
C01692=1060.986,-13.653,-67.311,171.642,27.542,155.124
C01693=1060.980,-13.902,-67.296,171.641,27.540,155.124
C01694=1060.974,-14.152,-67.283,171.639,27.538,155.124
C01695=1060.968,-14.401,-67.269,171.637,27.535,155.124
C01696=1060.962,-14.652,-67.255,171.636,27.533,155.123
C01697=1060.956,-14.900,-67.241,171.634,27.531,155.123
C01698=1060.950,-15.150,-67.227,171.633,27.529,155.123
C01699=1060.943,-15.400,-67.213,171.631,27.526,155.122
C01700=1060.938,-15.649,-67.199,171.629,27.524,155.122
C01701=1060.932,-15.899,-67.186,171.628,27.522,155.122
C01702=1060.925,-16.149,-67.173,171.626,27.519,155.122
C01703=1060.919,-16.398,-67.158,171.625,27.517,155.121
C01704=1060.913,-16.647,-67.145,171.624,27.515,155.121
C01705=1060.907,-16.897,-67.130,171.622,27.513,155.121
C01706=1060.901,-17.146,-67.117,171.621,27.511,155.121
C01707=1060.894,-17.396,-67.104,171.619,27.509,155.120
C01708=1060.888,-17.646,-67.090,171.617,27.507,155.120
C01709=1060.881,-17.925,-67.074,171.616,27.504,155.120
C01710=1060.874,-18.204,-67.059,171.613,27.501,155.120
C01711=1060.868,-18.484,-67.044,171.612,27.499,155.119
C01712=1060.860,-18.764,-67.028,171.610,27.497,155.119
C01713=1060.854,-19.013,-67.015,171.609,27.494,155.119
C01714=1060.849,-19.263,-67.001,171.607,27.492,155.118
C01715=1060.842,-19.513,-66.987,171.605,27.490,155.118
C01716=1060.837,-19.762,-66.974,171.604,27.488,155.118
C01717=1060.830,-20.012,-66.960,171.602,27.485,155.118
C01718=1060.824,-20.260,-66.946,171.601,27.483,155.117
C01719=1060.818,-20.510,-66.932,171.599,27.481,155.117
C01720=1060.811,-20.760,-66.919,171.597,27.479,155.117
C01721=1060.805,-21.009,-66.906,171.597,27.477,155.117
C01722=1060.799,-21.259,-66.891,171.595,27.474,155.116
C01723=1060.793,-21.509,-66.878,171.593,27.473,155.116
C01724=1060.788,-21.758,-66.864,171.592,27.470,155.116
C01725=1060.781,-22.007,-66.851,171.590,27.468,155.116
C01726=1060.774,-22.257,-66.837,171.589,27.466,155.115
C01727=1060.769,-22.507,-66.823,171.587,27.464,155.115
C01728=1060.763,-22.756,-66.810,171.585,27.461,155.115
C01729=1060.757,-23.006,-66.798,171.584,27.459,155.115
C01730=1060.751,-23.256,-66.784,171.582,27.457,155.114
C01731=1060.745,-23.506,-66.770,171.581,27.454,155.114
C01732=1060.738,-23.755,-66.757,171.579,27.453,155.114
C01733=1060.733,-24.004,-66.743,171.577,27.450,155.114
C01734=1060.727,-24.254,-66.730,171.576,27.448,155.113
C01735=1060.720,-24.504,-66.716,171.574,27.446,155.113
C01736=1060.714,-24.753,-66.702,171.573,27.444,155.113
C01737=1060.708,-25.003,-66.689,171.571,27.441,155.113
C01738=1060.702,-25.252,-66.676,171.569,27.439,155.112
C01739=1060.696,-25.501,-66.662,171.568,27.437,155.112
C01740=1060.690,-25.751,-66.649,171.566,27.435,155.112
C01741=1060.684,-26.001,-66.636,171.564,27.433,155.112
C01742=1060.678,-26.251,-66.622,171.563,27.431,155.111
C01743=1060.672,-26.500,-66.608,171.561,27.428,155.111
C01744=1060.666,-26.749,-66.595,171.560,27.426,155.111
C01745=1060.660,-26.999,-66.582,171.559,27.424,155.110
C01746=1060.653,-27.249,-66.568,171.557,27.422,155.110
C01747=1060.648,-27.499,-66.555,171.556,27.420,155.110
C01748=1060.641,-27.748,-66.542,171.554,27.418,155.110
C01749=1060.635,-27.997,-66.529,171.552,27.416,155.110
C01750=1060.629,-28.247,-66.515,171.551,27.414,155.109
C01751=1060.622,-28.496,-66.502,171.549,27.412,155.109
C01752=1060.616,-28.746,-66.489,171.548,27.409,155.109
C01753=1060.610,-28.996,-66.476,171.546,27.408,155.109
C01754=1060.604,-29.245,-66.463,171.544,27.405,155.108
C01755=1060.598,-29.494,-66.449,171.543,27.403,155.108
C01756=1060.592,-29.745,-66.436,171.541,27.401,155.108
C01757=1060.586,-29.994,-66.423,171.539,27.399,155.108
C01758=1060.579,-30.244,-66.409,171.538,27.397,155.107
C01759=1060.574,-30.493,-66.397,171.536,27.395,155.107
C01760=1060.567,-30.743,-66.383,171.535,27.393,155.107
C01761=1060.561,-30.992,-66.370,171.533,27.391,155.107
C01762=1060.555,-31.241,-66.357,171.531,27.388,155.107
C01763=1060.548,-31.492,-66.344,171.530,27.387,155.106
C01764=1060.542,-31.741,-66.331,171.528,27.384,155.106
C01765=1060.536,-31.990,-66.317,171.527,27.382,155.106
C01766=1060.530,-32.240,-66.305,171.525,27.380,155.106
C01767=1060.524,-32.490,-66.292,171.523,27.378,155.105
C01768=1060.518,-32.739,-66.278,171.522,27.376,155.105
C01769=1060.512,-32.989,-66.265,171.520,27.374,155.105
C01770=1060.506,-33.238,-66.252,171.518,27.372,155.105
C01771=1060.500,-33.489,-66.239,171.517,27.369,155.104
C01772=1060.494,-33.738,-66.226,171.515,27.368,155.104
C01773=1060.487,-34.016,-66.212,171.514,27.366,155.104
C01774=1060.480,-34.295,-66.197,171.512,27.363,155.104
C01775=1060.473,-34.574,-66.182,171.509,27.361,155.104
C01776=1060.466,-34.852,-66.168,171.508,27.358,155.103
C01777=1060.460,-35.102,-66.155,171.506,27.356,155.103
C01778=1060.454,-35.351,-66.142,171.505,27.354,155.103
C01779=1060.448,-35.601,-66.129,171.503,27.352,155.103
C01780=1060.442,-35.851,-66.116,171.501,27.350,155.102
C01781=1060.436,-36.101,-66.103,171.500,27.348,155.102
C01782=1060.429,-36.350,-66.090,171.498,27.346,155.102
C01783=1060.424,-36.600,-66.078,171.496,27.344,155.102
C01784=1060.417,-36.849,-66.064,171.495,27.342,155.102
C01785=1060.412,-37.099,-66.051,171.493,27.340,155.101
C01786=1060.406,-37.348,-66.038,171.491,27.338,155.101
C01787=1060.400,-37.598,-66.025,171.490,27.336,155.101
C01788=1060.394,-37.848,-66.012,171.488,27.333,155.101
C01789=1060.388,-38.097,-65.999,171.487,27.332,155.100
C01790=1060.382,-38.347,-65.986,171.485,27.329,155.100
C01791=1060.376,-38.597,-65.974,171.483,27.328,155.100
C01792=1060.369,-38.846,-65.961,171.482,27.325,155.100
C01793=1060.363,-39.095,-65.948,171.480,27.324,155.100
C01794=1060.356,-39.345,-65.935,171.478,27.321,155.099
C01795=1060.350,-39.595,-65.922,171.477,27.320,155.099
C01796=1060.344,-39.845,-65.910,171.475,27.317,155.099
C01797=1060.338,-40.094,-65.896,171.474,27.316,155.099
C01798=1060.331,-40.344,-65.884,171.472,27.313,155.099
C01799=1060.325,-40.593,-65.871,171.470,27.312,155.098
C01800=1060.319,-40.843,-65.859,171.469,27.309,155.098
C01801=1060.313,-41.093,-65.846,171.467,27.308,155.098
C01802=1060.307,-41.342,-65.833,171.465,27.306,155.098
C01803=1060.301,-41.592,-65.821,171.464,27.304,155.098
C01804=1060.295,-41.842,-65.808,171.462,27.302,155.097
C01805=1060.288,-42.091,-65.795,171.460,27.300,155.097
C01806=1060.283,-42.341,-65.782,171.459,27.298,155.097
C01807=1060.276,-42.590,-65.770,171.457,27.296,155.097
C01808=1060.270,-42.840,-65.757,171.455,27.294,155.097
C01809=1060.264,-43.090,-65.745,171.454,27.292,155.096
C01810=1060.258,-43.339,-65.732,171.452,27.290,155.096
C01811=1060.252,-43.589,-65.719,171.451,27.288,155.096
C01812=1060.245,-43.838,-65.707,171.449,27.286,155.096
C01813=1060.239,-44.088,-65.694,171.447,27.284,155.096
